// TIA Portal project "main" (V14)

(* hardware
DEVICE "GSD-Geraet_1"  GSD.Device.PN
   slot 0: "Baugruppenträger"  Rail  V1.0
   slot 0: "Station1"  BNI005H  V3.0
   slot 4: "SmartLight2"  IOL_I/O_08/08 byte
      slot 0: "IOL_I/O_08/08 byte"  IOL_I/O_08/08 byte
DEVICE "ET 200SP-Station_2"  ET 200SP-Station
   slot 0: "Baugruppenträger_0"  6ES5 710-8MAx1
   slot 1: "PLC_1"  CPU 1512SP F-1 PN  6ES7 512-1SK01-0AB0  V2.0
   slot 2: "DI 8x24VDC HF_1"  DI 8x24VDC HF  6ES7 131-6BF00-0CA0  V1.2
      slot 1: "DI 8x24VDC HF_1"  DI 8x24VDC HF
   slot 3: "Servermodul_1"  Servermodul  6ES7 193-6PA00-0AA0  V1.0
      slot 1: "Servermodul_1"  Servermodul
   slot 127: "BA 2xRJ45"  BA 2xRJ45  6ES7 193-6AR00-0AA0  V0.0
      slot 32769: "Port_1"  6ES7 193-6AR00-0AA0
      slot 32770: "Port_2"  6ES7 193-6AR00-0AA0
DEVICE "GSD-Geraet_2"  GSD.Device.PN
   slot 0: "Baugruppenträger"  Rail  V1.0
   slot 0: "Station2"  BNI005H  V3.0
DEVICE "GSD-Geraet_3"  GSD.Device.PN
   slot 0: "Baugruppenträger"  Rail  V1.0
   slot 0: "Station3"  BNI005H  V3.0
DEVICE "GSD-Geraet_4"  GSD.Device.PN
   slot 0: "Baugruppenträger"  Rail  V1.0
   slot 0: "Station4"  BNI005H  V3.0
   slot 4: "IOL_I/O_16/16 byte_3"  IOL_I/O_16/16 byte
      slot 0: "IOL_I/O_16/16 byte"  IOL_I/O_16/16 byte
DEVICE "GSD-Geraet_5"  GSD.Device.PN
   slot 0: "Baugruppenträger"  Rail  V1.0
   slot 0: "Station6"  BNI005H  V3.0
DEVICE "GSD-Geraet_6"  GSD.Device.PN
   slot 0: "Baugruppenträger"  Rail  V1.0
   slot 0: "Station8"  BNI005H  V3.0
   slot 3: "IOL_I/O_16/16 byte_2"  IOL_I/O_16/16 byte
      slot 0: "IOL_I/O_16/16 byte"  IOL_I/O_16/16 byte
   slot 4: "SmartLight"  IOL_I/O_08/08 byte
      slot 0: "IOL_I/O_08/08 byte"  IOL_I/O_08/08 byte
DEVICE "GSD-Geraet_7"  GSD.Device.PN
   slot 0: "Baugruppenträger"  Rail  V1.0
   slot 0: "Station7"  BNI005H  V3.0
DEVICE "GSD-Geraet_8"  GSD.Device.PN
   slot 0: "Baugruppenträger"  Rail  V1.0
   slot 0: "Station5"  BNI005H  V3.0
DEVICE "GSD-Geraet_9"  GSD.Device.PN
   slot 0: "Baugruppenträger"  Rail  V1.0
   slot 0: "Station10"  BNI005H  V3.0
DEVICE "GSD-Geraet_10"  GSD.Device.PN
   slot 0: "Baugruppenträger"  Rail  V1.0
   slot 0: "Station9"  BNI005H  V3.0
   slot 3: "IOL_I/O_16/16 byte_2"  IOL_I/O_16/16 byte
      slot 0: "IOL_I/O_16/16 byte"  IOL_I/O_16/16 byte
DEVICE "GSD-Geraet_11"  GSD.Device.PN
   slot 0: "Baugruppenträger"  Rail  V1.0
   slot 0: "Station11"  BNI005H  V3.0
   slot 4: "SmartLight2"  IOL_I/O_08/08 byte
      slot 0: "IOL_I/O_08/08 byte"  IOL_I/O_08/08 byte
DEVICE "GSD-Geraet_12"  GSD.Device.PN
   slot 0: "Baugruppenträger"  Rail  V1.0
   slot 0: "Station12"  BNI005H  V3.0
DEVICE "GSD-Geraet_13"  GSD.Device.PN
   slot 0: "Baugruppenträger"  Rail  V1.0
   slot 0: "Station13"  BNI005H  V3.0
DEVICE "GSD-Geraet_14"  GSD.Device.PN
   slot 0: "Baugruppenträger"  Rail  V1.0
   slot 0: "Station15"  BNI005H  V3.0
DEVICE "GSD-Geraet_15"  GSD.Device.PN
   slot 0: "Baugruppenträger"  Rail  V1.0
   slot 0: "Station16"  BNI005H  V3.0
DEVICE "GSD-Geraet_16"  GSD.Device.PN
   slot 0: "Baugruppenträger"  Rail  V1.0
   slot 0: "Station17"  BNI005H  V3.0
DEVICE "GSD-Geraet_17"  GSD.Device.PN
   slot 0: "Baugruppenträger"  Rail  V1.0
   slot 0: "Station20"  BNI005H  V3.0
DEVICE "GSD-Geraet_18"  GSD.Device.PN
   slot 0: "Baugruppenträger"  Rail  V1.0
   slot 0: "Station19"  BNI005H  V3.0
   slot 3: "IOL_I/O_16/16 byte_2"  IOL_I/O_16/16 byte
      slot 0: "IOL_I/O_16/16 byte"  IOL_I/O_16/16 byte
DEVICE "GSD-Geraet_19"  GSD.Device.PN
   slot 0: "Baugruppenträger"  Rack  V1.0
   slot 0: "BVS-SC"  BVS-SC  BVS_SC  V1.x
      slot 0: "BVS-SC"  BVS-SC
      slot 1: "PN-IO"  PN-IO
         slot 1: "port 1 - M12"  port 1 - M12
   slot 1: "SmartCamera E/A 128/16 Byte_1"  SmartCamera I/O 128/16 byte
      slot 0: "SmartCamera E/A 128/16 Byte"  SmartCamera I/O 128/16 byte
*)

// ===== PLC "PLC_1"  CPU 1512SP F-1 PN =====

VAR_GLOBAL   // PLC tag table "Standard-Variablentabelle"
   "EingangM1P1" AT %I1001.0 : Bool;
   "ByteM1P1.1" AT %IB1002 : Byte;
   "ByteM1P1.2" AT %IB1003 : Byte;
   "ByteM1P1.3" AT %IB1004 : Byte;
   "ByteM1P1.4" AT %IB1005 : Byte;
   "ByteM1P1.5" AT %IB1006 : Byte;
   "ByteM1P1.6" AT %IB1007 : Byte;
   "ByteM1P1.7" AT %IB1008 : Byte;
   "ByteM1P1.8" AT %IB1009 : Byte;
   "ByteM2P1.1" AT %IB2002 : Byte;
   "ByteM2P1.2" AT %IB2003 : Byte;
   "ByteM2P1.3" AT %IB2004 : Byte;
   "ByteM2P1.4" AT %IB2005 : Byte;
   "ByteM2P1.5" AT %IB2006 : Byte;
   "ByteM2P1.6" AT %IB2007 : Byte;
   "ByteM2P1.7" AT %IB2008 : Byte;
   "ByteM2P1.8" AT %IB2009 : Byte;
   "EingangM2P1" AT %I2001.0 : Bool;
   "ByteM3P1.1" AT %IB3002 : Byte;
   "ByteM3P1.2" AT %IB3003 : Byte;
   "ByteM3P1.3" AT %IB3004 : Byte;
   "ByteM3P1.4" AT %IB3005 : Byte;
   "ByteM3P1.5" AT %IB3006 : Byte;
   "ByteM3P1.6" AT %IB3007 : Byte;
   "ByteM3P1.7" AT %IB3008 : Byte;
   "ByteM3P1.8" AT %IB3009 : Byte;
   "EingangM3P1" AT %I3001.0 : Bool;
   "ByteM4P1.1" AT %IB4002 : Byte;
   "ByteM4P1.2" AT %IB4003 : Byte;
   "ByteM4P1.3" AT %IB4004 : Byte;
   "ByteM4P1.4" AT %IB4005 : Byte;
   "ByteM4P1.5" AT %IB4006 : Byte;
   "ByteM4P1.6" AT %IB4007 : Byte;
   "ByteM4P1.7" AT %IB4008 : Byte;
   "ByteM4P1.8" AT %IB4009 : Byte;
   "EingangM4P1" AT %I4001.0 : Bool;
   "ByteM5P1.1" AT %IB5002 : Byte;
   "ByteM5P1.2" AT %IB5003 : Byte;
   "ByteM5P1.3" AT %IB5004 : Byte;
   "ByteM5P1.4" AT %IB5005 : Byte;
   "ByteM5P1.5" AT %IB5006 : Byte;
   "ByteM5P1.6" AT %IB5007 : Byte;
   "ByteM5P1.7" AT %IB5008 : Byte;
   "ByteM5P1.8" AT %IB5009 : Byte;
   "EingangM5P1" AT %I5001.0 : Bool;
   "ByteM6P1.1" AT %IB6002 : Byte;
   "ByteM6P1.2" AT %IB6003 : Byte;
   "ByteM6P1.3" AT %IB6004 : Byte;
   "ByteM6P1.4" AT %IB6005 : Byte;
   "ByteM6P1.5" AT %IB6006 : Byte;
   "ByteM6P1.6" AT %IB6007 : Byte;
   "ByteM6P1.7" AT %IB6008 : Byte;
   "ByteM6P1.8" AT %IB6009 : Byte;
   "EingangM6P1" AT %I6001.0 : Bool;
   "ByteM7P1.1" AT %IB7002 : Byte;
   "ByteM7P1.2" AT %IB7003 : Byte;
   "ByteM7P1.3" AT %IB7004 : Byte;
   "ByteM7P1.4" AT %IB7005 : Byte;
   "ByteM7P1.5" AT %IB7006 : Byte;
   "ByteM7P1.6" AT %IB7007 : Byte;
   "ByteM7P1.7" AT %IB7008 : Byte;
   "ByteM7P1.8" AT %IB7009 : Byte;
   "EingangM7P1" AT %I7001.0 : Bool;
   "ByteM8P1.1" AT %IB8002 : Byte;
   "ByteM8P1.2" AT %IB8003 : Byte;
   "ByteM8P1.3" AT %IB8004 : Byte;
   "ByteM8P1.4" AT %IB8005 : Byte;
   "ByteM8P1.5" AT %IB8006 : Byte;
   "ByteM8P1.6" AT %IB8007 : Byte;
   "ByteM8P1.7" AT %IB8008 : Byte;
   "ByteM8P1.8" AT %IB8009 : Byte;
   "EingangM8P1" AT %I8001.0 : Bool;
   "ByteM9P1.1" AT %IB9002 : Byte;
   "ByteM9P1.2" AT %IB9003 : Byte;
   "ByteM9P1.3" AT %IB9004 : Byte;
   "ByteM9P1.4" AT %IB9005 : Byte;
   "ByteM9P1.5" AT %IB9006 : Byte;
   "ByteM9P1.6" AT %IB9007 : Byte;
   "ByteM9P1.7" AT %IB9008 : Byte;
   "ByteM9P1.8" AT %IB9009 : Byte;
   "EingangM9P1" AT %I9001.0 : Bool;
   "ByteM10P1.1" AT %IB10002 : Byte;
   "ByteM10P1.2" AT %IB10003 : Byte;
   "ByteM10P1.3" AT %IB10004 : Byte;
   "ByteM10P1.4" AT %IB10005 : Byte;
   "ByteM10P1.5" AT %IB10006 : Byte;
   "ByteM10P1.6" AT %IB10007 : Byte;
   "ByteM10P1.7" AT %IB10008 : Byte;
   "ByteM10P1.8" AT %IB10009 : Byte;
   "EingangM10P1" AT %I10001.0 : Bool;
   "ByteM11P1.1" AT %IB11002 : Byte;
   "ByteM11P1.2" AT %IB11003 : Byte;
   "ByteM11P1.3" AT %IB11004 : Byte;
   "ByteM11P1.4" AT %IB11005 : Byte;
   "ByteM11P1.5" AT %IB11006 : Byte;
   "ByteM11P1.6" AT %IB11007 : Byte;
   "ByteM11P1.7" AT %IB11008 : Byte;
   "ByteM11P1.8" AT %IB11009 : Byte;
   "EingangM11P1" AT %I11001.0 : Bool;
   "ByteM12P1.1" AT %IB12002 : Byte;
   "ByteM12P1.2" AT %IB12003 : Byte;
   "ByteM12P1.3" AT %IB12004 : Byte;
   "ByteM12P1.4" AT %IB12005 : Byte;
   "ByteM12P1.5" AT %IB12006 : Byte;
   "ByteM12P1.6" AT %IB12007 : Byte;
   "ByteM12P1.7" AT %IB12008 : Byte;
   "ByteM12P1.8" AT %IB12009 : Byte;
   "EingangM12P1" AT %I12001.0 : Bool;
   "ByteM13P1.1" AT %IB13002 : Byte;
   "ByteM13P1.2" AT %IB13003 : Byte;
   "ByteM13P1.3" AT %IB13004 : Byte;
   "ByteM13P1.4" AT %IB13005 : Byte;
   "ByteM13P1.5" AT %IB13006 : Byte;
   "ByteM13P1.6" AT %IB13007 : Byte;
   "ByteM13P1.7" AT %IB13008 : Byte;
   "ByteM13P1.8" AT %IB13009 : Byte;
   "EingangM13P1" AT %I13001.0 : Bool;
   "ByteM15P1.1" AT %IB15002 : Byte;
   "ByteM15P1.2" AT %IB15003 : Byte;
   "ByteM15P1.3" AT %IB15004 : Byte;
   "ByteM15P1.4" AT %IB15005 : Byte;
   "ByteM15P1.5" AT %IB15006 : Byte;
   "ByteM15P1.6" AT %IB15007 : Byte;
   "ByteM15P1.7" AT %IB15008 : Byte;
   "ByteM15P1.8" AT %IB15009 : Byte;
   "EingangM15P1" AT %I15001.0 : Bool;
   "ByteM16P1.1" AT %IB16002 : Byte;
   "ByteM16P1.2" AT %IB16003 : Byte;
   "ByteM16P1.3" AT %IB16004 : Byte;
   "ByteM16P1.4" AT %IB16005 : Byte;
   "ByteM16P1.5" AT %IB16006 : Byte;
   "ByteM16P1.6" AT %IB16007 : Byte;
   "ByteM16P1.7" AT %IB16008 : Byte;
   "ByteM16P1.8" AT %IB16009 : Byte;
   "EingangM16P1" AT %I16001.0 : Bool;
   "ByteM17P1.1" AT %IB17002 : Byte;
   "ByteM17P1.2" AT %IB17003 : Byte;
   "ByteM17P1.3" AT %IB17004 : Byte;
   "ByteM17P1.4" AT %IB17005 : Byte;
   "ByteM17P1.5" AT %IB17006 : Byte;
   "ByteM17P1.6" AT %IB17007 : Byte;
   "ByteM17P1.7" AT %IB17008 : Byte;
   "ByteM17P1.8" AT %IB17009 : Byte;
   "EingangM17P1" AT %I17001.0 : Bool;
   "ByteM19P1.1" AT %IB19002 : Byte;
   "ByteM19P1.2" AT %IB19003 : Byte;
   "ByteM19P1.3" AT %IB19004 : Byte;
   "ByteM19P1.4" AT %IB19005 : Byte;
   "ByteM19P1.5" AT %IB19006 : Byte;
   "ByteM19P1.6" AT %IB19007 : Byte;
   "ByteM19P1.7" AT %IB19008 : Byte;
   "ByteM19P1.8" AT %IB19009 : Byte;
   "EingangM19P1" AT %I19001.0 : Bool;
   "ByteM20P1.1" AT %IB20002 : Byte;
   "ByteM20P1.2" AT %IB20003 : Byte;
   "ByteM20P1.3" AT %IB20004 : Byte;
   "ByteM20P1.4" AT %IB20005 : Byte;
   "ByteM20P1.5" AT %IB20006 : Byte;
   "ByteM20P1.6" AT %IB20007 : Byte;
   "ByteM20P1.7" AT %IB20008 : Byte;
   "ByteM20P1.8" AT %IB20009 : Byte;
   "EingangM20P1" AT %I20001.0 : Bool;
   "EingangM4P2" AT %I4017.0 : Bool;
   "EingangM8P2" AT %I8017.0 : Bool;
   "ByteM8P2.1" AT %IB8018 : Byte;
   "ByteM8P2.2" AT %IB8019 : Byte;
   "ByteM8P2.3" AT %IB8020 : Byte;
   "ByteM8P2.4" AT %IB8021 : Byte;
   "ByteM8P2.5" AT %IB8022 : Byte;
   "ByteM8P2.6" AT %IB8023 : Byte;
   "ByteM8P2.7" AT %IB8024 : Byte;
   "ByteM8P2.8" AT %IB8025 : Byte;
   "EingangM9P2" AT %I9017.0 : Bool;
   "ByteM9P2.1" AT %IB9018 : Byte;
   "ByteM9P2.2" AT %IB9019 : Byte;
   "ByteM9P2.3" AT %IB9020 : Byte;
   "ByteM9P2.4" AT %IB9021 : Byte;
   "ByteM9P2.5" AT %IB9022 : Byte;
   "ByteM9P2.6" AT %IB9023 : Byte;
   "ByteM9P2.7" AT %IB9024 : Byte;
   "ByteM9P2.8" AT %IB9025 : Byte;
   "EingangM19P2" AT %I19017.0 : Bool;
   "ByteM19P2.1" AT %IB19018 : Byte;
   "ByteM19P2.2" AT %IB19019 : Byte;
   "ByteM19P2.3" AT %IB19020 : Byte;
   "ByteM19P2.4" AT %IB19021 : Byte;
   "ByteM19P2.5" AT %IB19022 : Byte;
   "ByteM19P2.6" AT %IB19023 : Byte;
   "ByteM19P2.7" AT %IB19024 : Byte;
   "ByteM19P2.8" AT %IB19025 : Byte;
   "EingangM4P2_AE" AT %I4017.2 : Bool;
   "EingangM4P3" AT %I4033.0 : Bool;
   "OutByteM1P2.1" AT %QB1017 : Byte;
   "BuzzerSmLi1" AT %Q1019.7 : Bool;
   "OutByteM4P2.1" AT %QB4018 : Byte;
   "OutHeader1M4P2_AV" AT %Q4017.0 : Bool;
   "OutByteM4P2.8" AT %QB4025 : Byte;
   "OutByteM4P2.7" AT %QB4024 : Byte;
   "OutByteM4P2.6" AT %QB4023 : Byte;
   "OutByteM4P2.5" AT %QB1022 : Byte;
   "OutByteM4P2.4" AT %QB4021 : Byte;
   "OutByteM4P2.3" AT %QB4020 : Byte;
   "OutByteM4P2.2" AT %QB4019 : Byte;
   "OutHeader2M4P2_AV" AT %Q4026.0 : Bool;
   "OutByteM1P3_Level8bit" AT %QB1027 : Byte;
   "SmLiS1P3-0.0" AT %Q1021.0 : Bool;
   "SmLiS1P3-0.1" AT %Q1021.1 : Bool;
   "SmLiS1P3-0.2" AT %Q1021.2 : Bool;
   "SmLiS1P3-0.3" AT %Q1021.3 : Bool;
   "SmLiS1P3-0.4" AT %Q1021.4 : Bool;
   "SmLiS1P3-0.5" AT %Q1021.5 : Bool;
   "SmLiS1P3-0.6" AT %Q1021.6 : Bool;
   "SmLiS1P3-0.7" AT %Q1021.7 : Bool;
   "SmLiS1P3-1.0" AT %Q1022.0 : Bool;
   "SmLiS1P3-1.1" AT %Q1022.1 : Bool;
   "SmLiS1P3-1.3" AT %Q1022.3 : Bool;
   "SmLiS1P3-1.4" AT %Q1022.4 : Bool;
   "SmLiS1P3-1.5" AT %Q1022.5 : Bool;
   "SmLiS1P3-1.6" AT %Q1022.6 : Bool;
   "SmLiS1P3-1.2" AT %Q1022.2 : Bool;
   "SmLiS1P3-1.7" AT %Q1022.7 : Bool;
   "SmLiS1P3-2.3" AT %Q1023.3 : Bool;
   "SmLiS1P3-2.2" AT %Q1023.2 : Bool;
   "SmLiS1P3-2.1" AT %Q1023.1 : Bool;
   "SmLiS1P3-2.0" AT %Q1023.0 : Bool;
   "SmLiS1P3-3.1-Levelmode" AT %Q1024.1 : Bool;
   "OutByteM11P2.1" AT %QB11017 : Byte;
   "OutByteM11P3_Level8bit" AT %QB11027 : Byte;
   "SmLiS11P3-0.0" AT %Q11021.0 : Bool;
   "SmLiS11P3-0.1" AT %Q11021.1 : Bool;
   "SmLiS11P3-0.2" AT %Q11021.2 : Bool;
   "SmLiS11P3-0.3" AT %Q11021.3 : Bool;
   "SmLiS11P3-0.4" AT %Q11021.4 : Bool;
   "SmLiS11P3-0.5" AT %Q11021.5 : Bool;
   "SmLiS11P3-0.6" AT %Q11021.6 : Bool;
   "SmLiS11P3-0.7" AT %Q11021.7 : Bool;
   "SmLiS11P3-1.0" AT %Q11022.0 : Bool;
   "SmLiS11P3-1.1" AT %Q11022.1 : Bool;
   "SmLiS11P3-1.2" AT %Q11022.2 : Bool;
   "SmLiS11P3-1.3" AT %Q11022.3 : Bool;
   "SmLiS11P3-1.4" AT %Q11022.4 : Bool;
   "SmLiS11P3-1.5" AT %Q11022.5 : Bool;
   "SmLiS11P3-1.6" AT %Q11022.6 : Bool;
   "SmLiS11P3-1.7" AT %Q11022.7 : Bool;
   "SmLiS11P3-2.0" AT %Q11023.0 : Bool;
   "SmLiS11P3-2.1" AT %Q11023.1 : Bool;
   "SmLiS11P3-2.2" AT %Q11023.2 : Bool;
   "SmLiS11P3-2.3" AT %Q11023.3 : Bool;
   "SmLiS11P3-3.1-Levelmode" AT %Q11024.1 : Bool;
   "SmLiS8P3-0.0" AT %Q8033.0 : Bool;
   "SmLiS8P3-0.1" AT %Q8033.1 : Bool;
   "SmLiS8P3-0.4" AT %Q8033.4 : Bool;
   "SmLiS8P3-0.5" AT %Q8033.5 : Bool;
   "SmLiS8P3-1.0" AT %Q8034.0 : Bool;
   "SmLiS8P3-1.1" AT %Q8034.1 : Bool;
   "SmLiS8P3-1.4" AT %Q8034.4 : Bool;
   "SmLiS8P3-1.5" AT %Q8034.5 : Bool;
   "SmLiS8P3-2.0" AT %Q8035.0 : Bool;
   "SmLiS8P3-2.1" AT %Q8035.1 : Bool;
   "SmLiS8P3-3.0-Segmentmode" AT %Q8036.0 : Bool;
   "Clock" AT %M0.0 : Bool;
   "inPuffer" AT %MB100 : Byte;
   "ausPuffer" AT %MB2 : Byte;
   "Testmerker1" AT %M0.1 : Bool;
   "SC_CommandStart" AT %M0.2 : Bool;
   "SC_CamResetWarn" AT %M200.0 : Bool;
   "SC_GetResults" AT %M0.7 : Bool;
   "SC_Trigger" AT %M0.6 : Bool;
   "SC_StartRun" AT %M0.5 : Bool;
   "SC_StopRun" AT %M0.4 : Bool;
   "SC_ResetWarnings" AT %M0.3 : Bool;
   "MerkerCommandSC" AT %MW201 : Int;
   "S9P1IB0.2_AE" AT %I9001.2 : Bool;
   "S9P1IB0.1_AA" AT %I9001.1 : Bool;
   "S9P1OB0.0_AV" AT %Q9001.0 : Bool;
   "S9P1OB1_CommandDesignator" AT %QB9002 : Byte;
   "S9P1OB2_StartAdressLow" AT %QB9003 : Byte;
   "S9P1OB3_StartAdressHigh" AT %QB9004 : Byte;
   "S9P1OB4_NumBytesLow" AT %QB9005 : Byte;
   "S9P1OB5_NumBytesHigh" AT %QB9006 : Byte;
   "S9P1OB9.0_AV" AT %Q9010.0 : Bool;
   "S1P1OB1_CommandDesignator" AT %QB1002 : Byte;
   "S1P1OB2_StartAdressLow" AT %QB1003 : Byte;
   "S1P1OB3_StartAdressHigh" AT %QB1004 : Byte;
   "S1P1OB4_NumBytesLow" AT %QB1005 : Byte;
   "S1P1OB4_NumBytesHigh" AT %QB1006 : Byte;
   "S1P1OB0.0_AV" AT %Q1001.0 : Bool;
   "S1P1OB9.0_AV" AT %Q1010.0 : Bool;
   "S1P1IB0.2_AE" AT %Q1010.2 : Bool;
   "S1P1IB0.3_AF" AT %Q1010.3 : Bool;
   "S1P1IB0.1_AA" AT %Q1010.1 : Bool;
   "S9P2OB1_CommandDesignator" AT %QB9018 : Byte;
   "S9P2OB2_StartAdressLow" AT %QB9019 : Byte;
   "S9P2OB3_StartAdressHigh" AT %QB9020 : Byte;
   "S9P2OB4_NumBytesLow" AT %QB9021 : Byte;
   "S9P2OB4_NumBytesHigh" AT %QB9022 : Byte;
   "S9P2OB0.0_AV" AT %Q9017.0 : Bool;
   "S9P2OB9.0_AV" AT %Q9026.0 : Bool;
   "S9P2IB0.2_AE" AT %Q9017.2 : Bool;
   "S9P2IB0.3_AF" AT %Q9017.3 : Bool;
   "S9P2IB0.1_AA" AT %Q9017.1 : Bool;
   "ByteM4P2.1" AT %IB4018 : Byte;
   "ByteM4P2.2" AT %IB4019 : Byte;
   "ByteM4P2.3" AT %IB4020 : Byte;
   "ByteM4P2.4" AT %IB4021 : Byte;
   "ByteM4P2.5" AT %IB4022 : Byte;
   "ByteM4P2.6" AT %IB4023 : Byte;
   "ByteM4P2.7" AT %IB4024 : Byte;
   "ByteM4P2.8" AT %IB4025 : Byte;
   "ByteM4P3.1" AT %IB4034 : Byte;
   "ByteM4P3.2" AT %IB4035 : Byte;
   "ByteM4P3.3" AT %IB4036 : Byte;
   "ByteM4P3.4" AT %IB4037 : Byte;
   "ByteM4P3.5" AT %IB4038 : Byte;
   "ByteM4P3.6" AT %IB4039 : Byte;
   "ByteM4P3.7" AT %IB4040 : Byte;
   "ByteM4P3.8" AT %IB4041 : Byte;
   "Tag_1" AT %T1 : Timer;
END_VAR

DATA_BLOCK "IO_LINK_MASTER_DB"   // DB1
{ S7_Optimized_Access := 'TRUE' }
AUTHOR : Siemens
FAMILY : IO-Link
VERSION : 1.0
// stored: InstanceOfName IO_LINK_MASTER
"IO_LINK_MASTER"
BEGIN
END_DATA_BLOCK

DATA_BLOCK "IO_LINK_DEVICE_DB"   // DB2
{ S7_Optimized_Access := 'TRUE' }
AUTHOR : SUP_FA
FAMILY : IO-Link
VERSION : 3.0
// stored: InstanceOfName IO_LINK_DEVICE
"IO_LINK_DEVICE"
BEGIN
   write.data[0] := 16#03;
END_DATA_BLOCK

DATA_BLOCK "BVS_SC_DB"   // DB7
{ S7_Optimized_Access := 'TRUE' }
AUTHOR : BI-CU
FAMILY : Balluff
VERSION : 1.1
// stored: InstanceOfName BVS_SC
"BVS_SC"
BEGIN
END_DATA_BLOCK

DATA_BLOCK "00TEMP"   // DB8
{ S7_Optimized_Access := 'TRUE' }
VERSION : 0.1
   VAR
      EingriffPufferstand : Int;
      EingriffSmLiNummer : Int := 1;
      FlagEingriff : Bool;
      FlankenmerkerEingriff : Bool;
      Station1Umschaltung : Bool;
      TempAdresseFlag : Bool;
      RET_VAL : Int;
      PIADDR : UDInt;
      PICOUNT : UInt;
      PQADDR : UDInt;
      PQCOUNT : UInt;
      TempFlagPeek : Bool;
      ArrayTemp : Array[0..7] of Byte;
      ID : String;
      TempFlankenmerkePeek : Bool;
   END_VAR
BEGIN
END_DATA_BLOCK

DATA_BLOCK "FB35_Station1"   // DB11
{ S7_Optimized_Access := 'FALSE' }
AUTHOR : Serrano
FAMILY : Ident
NAME : BISM_IOL
VERSION : 1.0
// stored: InstanceOfName FB35_IOL_10Byte
"FB35_IOL_10Byte"
BEGIN
   Watchdog := S5T#3000MS;
END_DATA_BLOCK

DATA_BLOCK "Daten_zu_SC_Station8"   // DB12
{ S7_Optimized_Access := 'FALSE' }
VERSION : 0.1
   VAR
      SendByte : Array[0..99] of Byte;
   END_VAR
BEGIN
   SendByte[0] := 16#2;
   SendByte[1] := 16#0;
   SendByte[2] := 16#0;
   SendByte[3] := 16#0;
   SendByte[4] := 16#0;
END_DATA_BLOCK

DATA_BLOCK "Daten_von_SC_Station8"   // DB13
{ S7_Optimized_Access := 'FALSE' }
VERSION : 0.1
   VAR
      "n.u." : Byte;
      AppID : Byte;
      Buerstentraeger : Bool;
      "n.u._7" : Bool;
      "n.u._6" : Bool;
      "n.u._5" : Bool;
      "n.u._4" : Bool;
      "n.u._3" : Bool;
      "n.u._2" : Bool;
      "n.u._1" : Bool;
      GehaeuseUnten_Schraube : Bool;
      "n.u._14" : Bool;
      "n.u._13" : Bool;
      "n.u._12" : Bool;
      "n.u._11" : Bool;
      "n.u._10" : Bool;
      "n.u._9" : Bool;
      "n.u._8" : Bool;
      Zahnrad_klein : Bool;
      "n.u._21" : Bool;
      "n.u._20" : Bool;
      "n.u._19" : Bool;
      "n.u._18" : Bool;
      "n.u._17" : Bool;
      "n.u._16" : Bool;
      "n.u._15" : Bool;
      Zahnrad_gross : Bool;
      "n.u._28" : Bool;
      "n.u._27" : Bool;
      "n.u._26" : Bool;
      "n.u._25" : Bool;
      "n.u._24" : Bool;
      "n.u._23" : Bool;
      "n.u._22" : Bool;
      GehaeuseOben : Bool;
   END_VAR
BEGIN
END_DATA_BLOCK

DATA_BLOCK "DB_Ausfall_IO"   // DB16
{ S7_Optimized_Access := 'TRUE' }
VERSION : 0.1
   VAR
      ErrorCode_RD_SINFO : Int;
      ErrorCode_RD_SYS_T : Int;
      ErrorCode_LOG2GEO : Int;
      ErrorCode_D_ACT_DP : Int;
      ErrorCode_ModuleStates1 : Int;
      ErrorCode_ModuleStates2 : Int;
      StateBusy_D_ACT_DP : Bool;
      State1 : Array[0..127] of Bool;
      State2 : Array[0..127] of Bool;
      TimeOfEvent : DTL;
      FlagAdresseUmgewandelt : Bool;
      Info : SI_StationFailure;
      TempAdresse : Hw_Device;
      Info_2 : SI_classic;
      AdresseAusfall : GEOADDR;
      CounterS1 : Int;
      CounterS2 : Int;
      CounterS3 : Int;
      CounterS4 : Int;
      CounterS5 : Int;
      CounterS6 : Int;
      CounterS7 : Int;
      CounterS8 : Int;
      CounterS9 : Int;
      CounterS10 : Int;
      FlagDeaktivieren : Bool;
      bibop : Bool;
      ToggleNeu : Bool;
      CounterRack : Int;
      CounterStatus : Int;
      CounterProfile : Int;
      CounterPull : Int;
      CounterIO : Int;
      Adressen : Array[0..2] of HW_IO;
   END_VAR
BEGIN
END_DATA_BLOCK

DATA_BLOCK "Daten_von_SLK"   // DB17
{ S7_Optimized_Access := 'TRUE' }
VERSION : 0.1
   VAR
      V34 : Byte;
      V35 : Byte;
      V3 : Byte;
      V4 : Byte;
      V5 : Byte;
      V6 : Byte;
      V7 : Byte;
      V8 : Byte;
      V9 : Byte;
      V10 : Byte;
      V11 : Byte;
      V33 : Byte;
      V32 : Byte;
      V31 : Byte;
      V30 : Byte;
      V29 : Byte;
      V28 : Byte;
      V27 : Byte;
      V26 : Byte;
      V25 : Byte;
      V24 : Byte;
      V23 : Byte;
      V22 : Byte;
      V21 : Byte;
      V20 : Byte;
      V19 : Byte;
      V18 : Byte;
      V17 : Byte;
      V16 : Byte;
      V15 : Byte;
      V14 : Byte;
      V13 : Byte;
      V12 : Byte;
   END_VAR
BEGIN
END_DATA_BLOCK

DATA_BLOCK "Daten_zu_SLK"   // DB18
{ S7_Optimized_Access := 'TRUE' }
VERSION : 0.1
   VAR
      V11 : Byte;
      V34 : Byte;
      V33 : Byte;
      V32 : Byte;
      V31 : Byte;
      V30 : Byte;
      V29 : Byte;
      V28 : Byte;
      V27 : Byte;
      V26 : Byte;
      V25 : Byte;
      V24 : Byte;
      V23 : Byte;
      V22 : Byte;
      V21 : Byte;
      V20 : Byte;
      V19 : Byte;
      V18 : Byte;
      V17 : Byte;
      V16 : Byte;
      V15 : Byte;
      V14 : Byte;
      V13 : Byte;
      V12 : Byte;
   END_VAR
BEGIN
END_DATA_BLOCK

DATA_BLOCK "Lese_DB_1"   // DB19
{ S7_Optimized_Access := 'TRUE' }
VERSION : 0.1
// stored: InstanceOfName Lese
"Lese"
BEGIN
   Adresse := 1002;
   EndeAdresse := 1009;
END_DATA_BLOCK

DATA_BLOCK "DB_Konstanten"   // DB20
{ S7_Optimized_Access := 'TRUE' }
VERSION : 0.1
   VAR
      HW_Adressen : Array[0..19] of HW_ANY;
      "Anzahl Adressen" : Int := 20;
      DEFAULT_STATION4_MAXPUFFER : Array[0..1] of Int;
   END_VAR
BEGIN
   DEFAULT_STATION4_MAXPUFFER[1] := 19;
   DEFAULT_STATION4_MAXPUFFER[0] := 12;
END_DATA_BLOCK

DATA_BLOCK "Test"   // DB21
{ S7_Optimized_Access := 'TRUE' }
VERSION : 0.1
   VAR
      RetValD_ACT_DP2 : Int;
      RetValD_ACT_DP1 : Int;
      RetValD_ACT_DP3 : Int;
      RetValState1 : Int;
      RetValState2 : Int;
      Busy1 : Bool;
      Busy2 : Bool;
      Busy3 : Bool;
      State1 : Bool;
      State2 : Bool;
      Req : Bool;
      IstDeakt1 : Int;
      IstDeakt2 : Int;
      FlagDeak : Bool;
      FlagDeakAll1 : Bool;
      FlagDeakAll2 : Bool;
      FlagDeakAll3 : Bool;
      FlagDeakAll4 : Bool;
      FlagDeakAll5 : Bool;
      FlagAk : Bool;
   END_VAR
BEGIN
END_DATA_BLOCK

DATA_BLOCK "DB_Station1_Port1"   // DB101
{ S7_Optimized_Access := 'FALSE' }
VERSION : 0.1
   VAR
      TagAtHead : Bool;
      Station : Byte := 1;
      Port : Byte := 1;
      CurrentValue_ULInt : ULInt;
      CurrentValue : String;
      RET_VAL : Int := 0;
      Busy : Bool := false;
      Deactivated : Bool := false;
      State : Bool;
      State2 : Bool;
      RET_VAL_module_state : Int;
      IDRead : Bool;
      PoltopfLength : Byte;
      Flag : Bool;
      Done : Bool;
      TimeWaited : Time;
      TempFlagDeaktivierung : Bool;
      TEMPCounter : Int;
      S1P1FlankePos : Bool;
   END_VAR
BEGIN
END_DATA_BLOCK

DATA_BLOCK "DB_Station2_Port1"   // DB201
{ S7_Optimized_Access := 'FALSE' }
VERSION : 0.1
   VAR
      TagAtHead : Bool;
      Station : Byte := 2;
      Port : Byte := 1;
      CurrentValue_ULInt : ULInt := 0;
      CurrentValue : String := '';
      RET_VAL : Int := 0;
      Busy : Bool := false;
      Deactivated : Bool := false;
      State : Bool;
      State2 : Bool;
      RET_VAL_module_state : Int;
   END_VAR
BEGIN
END_DATA_BLOCK

DATA_BLOCK "DB_Station3_Port1"   // DB301
{ S7_Optimized_Access := 'FALSE' }
VERSION : 0.1
   VAR
      TagAtHead : Bool;
      Station : Byte := 3;
      Port : Byte := 1;
      CurrentValue_ULInt : ULInt := 0;
      CurrentValue : String := '';
      RET_VAL : Int := 0;
      Busy : Bool := false;
      Deactivated : Bool := false;
      State : Bool;
      State2 : Bool;
      RET_VAL_module_state : Int;
   END_VAR
BEGIN
END_DATA_BLOCK

DATA_BLOCK "DB_Station4_Port1"   // DB401
{ S7_Optimized_Access := 'FALSE' }
VERSION : 0.1
   VAR
      TagAtHead : Bool;
      Station : Byte := 4;
      Port : Byte := 1;
      CurrentValue_ULInt : ULInt := 0;
      CurrentValue : String := '';
      LastValue_ULInt : ULInt := 0;
      RET_VAL : Int := 0;
      Busy : Bool := false;
      Deactivated : Bool := false;
      State : Bool;
      State2 : Bool;
      RET_VAL_module_state : Int;
   END_VAR
BEGIN
END_DATA_BLOCK

DATA_BLOCK "DB_Station4_Puffer"   // DB410
{ S7_Optimized_Access := 'FALSE' }
VERSION : 0.1
   VAR
      CONST_MAXPUFFER : Array[0..1] of Int;
      CONST_STARTWERT_SMLI1 : Int := 0;
      Pufferstand : Array[0..1] of Int;
      Faktoren : Array[0..1] of Int;
      CurrentID1 : ULInt;
      LastID1 : ULInt;
      CurrentID2 : ULInt;
      LastID2 : ULInt;
      TimeRun1 : Time := T#5s;
      TimeRun2 : Time;
      FlankenmerkerPort1Pos : Bool;
      FlankenmerkerPort2Neg : Bool;
      FlankenmerkerPort3Neg : Bool;
      FlankenmerkerPort2Pos : Bool;
      FlankenmerkerPort3Pos : Bool;
      FlankenmerkerPosTime1 : Bool;
      FlankenmerkerPosTime2 : Bool;
      FlagTimerStart1 : Bool;
      FlagTimerStart2 : Bool;
      FlagShortcut1 : Bool;
      FlagShortcut2 : Bool;
      temp : Bool;
   END_VAR
BEGIN
   CONST_MAXPUFFER[0] := 12;
   CONST_MAXPUFFER[1] := 19;
   Faktoren[0] := 0;
   Faktoren[1] := 0;
END_DATA_BLOCK

DATA_BLOCK "DB_Station5_Port1"   // DB501
{ S7_Optimized_Access := 'FALSE' }
VERSION : 0.1
   VAR
      TagAtHead : Bool;
      Station : Byte := 5;
      Port : Byte := 1;
      CurrentValue_ULInt : ULInt := 0;
      CurrentValue : String := '';
      RET_VAL : Int := 0;
      Busy : Bool := false;
      Deactivated : Bool := false;
      State : Bool;
      State2 : Bool;
      RET_VAL_module_state : Int;
   END_VAR
BEGIN
END_DATA_BLOCK

DATA_BLOCK "DB_Station6_Port1"   // DB601
{ S7_Optimized_Access := 'FALSE' }
VERSION : 0.1
   VAR
      TagAtHead : Bool;
      Station : Byte := 6;
      Port : Byte := 1;
      CurrentValue_ULInt : ULInt := 0;
      CurrentValue : String := '';
      RET_VAL : Int := 0;
      Busy : Bool := false;
      Deactivated : Bool := false;
      State : Bool;
      State2 : Bool;
      RET_VAL_module_state : Int;
   END_VAR
BEGIN
END_DATA_BLOCK

DATA_BLOCK "DB_Station7_Port1"   // DB701
{ S7_Optimized_Access := 'FALSE' }
VERSION : 0.1
   VAR
      TagAtHead : Bool;
      Station : Byte := 7;
      Port : Byte := 1;
      CurrentValue_ULInt : ULInt := 0;
      CurrentValue : String := '';
      RET_VAL : Int := 0;
      Busy : Bool := false;
      Deactivated : Bool := false;
      State : Bool;
      State2 : Bool;
      RET_VAL_module_state : Int;
   END_VAR
BEGIN
END_DATA_BLOCK

DATA_BLOCK "DB_Station8_Port1"   // DB801
{ S7_Optimized_Access := 'FALSE' }
VERSION : 0.1
   VAR
      TagAtHead : Bool;
      Station : Byte := 8;
      Port : Byte := 1;
      CurrentValue_ULInt : ULInt := 0;
      CurrentValue : String := '';
      RET_VAL : Int := 0;
      RET_VAL_Camera : Int;
      Busy_Camera : Bool;
      Busy : Bool := false;
      Deactivated : Bool := false;
      State : Bool;
      State2 : Bool;
      RET_VAL_module_state : Int;
   END_VAR
BEGIN
END_DATA_BLOCK

DATA_BLOCK "DB_Station8_Port2"   // DB802
{ S7_Optimized_Access := 'FALSE' }
VERSION : 0.1
   VAR
      TagAtHead : Bool;
      Station : Byte := 8;
      Port : Byte := 2;
      CurrentValue_ULInt : ULInt := 0;
      CurrentValue : String := '';
   END_VAR
BEGIN
END_DATA_BLOCK

DATA_BLOCK "DB_SC_Station8"   // DB810
{ S7_Optimized_Access := 'TRUE' }
VERSION : 0.1
   VAR
      Buerstentraeger : Bool;
      GehaeuseUnten_Schraube : Bool;
      Zahnrad_klein : Bool;
      Zahnrad_gross : Bool;
      GehaeuseOben : Bool;
      FlankenmerkerP1 : Bool;
      FlankenmerkerP4 : Bool;
      FlankenmerkerP3 : Bool;
      FlankenmerkerP2 : Bool;
      FlankenmerkerGetResult1 : Bool;
      FlankenmerkerGetResult2 : Bool;
      setzezurüeck1 : Bool;
      setzezurüeck2 : Bool;
      startePruefung : Bool;
      CommandFlanke1 : Bool;
      StartRun_Flanke : Bool;
      ResetWarnings_Flanke : Bool;
      StopRun_Flanke : Bool;
      GetResult_Flanke : Bool;
      Trigger_Flanke : Bool;
      CamBusy_Flanke : Bool;
      Verzoegerung : Time;
   END_VAR
BEGIN
END_DATA_BLOCK

DATA_BLOCK "DB_Station9_Port1"   // DB901
{ S7_Optimized_Access := 'FALSE' }
VERSION : 0.1
   VAR
      TagAtHead : Bool;
      Station : Byte := 9;
      Port : Byte := 1;
      CurrentValue_ULInt : ULInt := 0;
      CurrentValue : String := '';
      RET_VAL : Int := 0;
      Busy : Bool := false;
      Deactivated : Bool := false;
      State : Bool;
      State2 : Bool;
      RET_VAL_module_state : Int;
      TriggerAltNeu : Bool := true;
      ToReadStartByteHigh : Byte := 16#0;
      ToReadStartByteLow : Byte;
      ToReadNumBytesLow : Byte := 16#1;
      ToReadNumBytesHigh : Byte;
      ReadByte1 : Byte := 16#27;
      ReadByte2 : Byte := 16#27;
      ReadByte3 : Byte := 16#27;
      ReadByte4 : Byte := 16#27;
      ReadByte5 : Byte := 16#27;
      ReadByte6 : Byte := 16#27;
      ReadByte7 : Byte := 16#27;
      ReadByte8 : Byte := 16#27;
      ErrorCode : Byte;
      FlagAngekommen_4 : Bool;
      FlagAngekommen_3 : Bool;
      FlagAngekommen_2 : Bool;
      FlagAngekommen_1 : Bool;
      FlagAngekommen : Bool;
   END_VAR
BEGIN
END_DATA_BLOCK

DATA_BLOCK "DB_Station9_Port2"   // DB902
{ S7_Optimized_Access := 'FALSE' }
VERSION : 0.1
   VAR
      TagAtHead : Bool;
      Station : Byte := 9;
      Port : Byte := 2;
      CurrentValue_ULInt : ULInt := 0;
      CurrentValue : String := '';
      IDRead : Bool;
      PoltopfLength : Byte;
      Flag : Bool;
      Done : Bool;
      TimeWaited : Time;
   END_VAR
BEGIN
END_DATA_BLOCK

DATA_BLOCK "DB_Station10_Port1"   // DB1001
{ S7_Optimized_Access := 'FALSE' }
VERSION : 0.1
   VAR
      TagAtHead : Bool;
      Station : Byte := 10;
      Port : Byte := 1;
      CurrentValue_ULInt : ULInt := 0;
      CurrentValue : String := '';
      RET_VAL : Int := 0;
      Busy : Bool := false;
      Deactivated : Bool := false;
      State : Bool;
      State2 : Bool;
      RET_VAL_module_state : Int;
   END_VAR
BEGIN
END_DATA_BLOCK

DATA_BLOCK "DB_Station11_Port1"   // DB1101
{ S7_Optimized_Access := 'FALSE' }
VERSION : 0.1
   VAR
      TagAtHead : Bool;
      Station : Byte := 11;
      Port : Byte := 1;
      CurrentValue_ULInt : ULInt := 0;
      CurrentValue : String := '';
      RET_VAL : Int := 0;
      Busy : Bool := false;
      Deactivated : Bool := false;
      State : Bool;
      State2 : Bool;
      RET_VAL_module_state : Int;
   END_VAR
BEGIN
END_DATA_BLOCK

DATA_BLOCK "DB_Station12_Port1"   // DB1201
{ S7_Optimized_Access := 'FALSE' }
VERSION : 0.1
   VAR
      TagAtHead : Bool;
      Station : Byte := 12;
      Port : Byte := 1;
      CurrentValue_ULInt : ULInt := 0;
      CurrentValue : String := '';
      RET_VAL : Int := 0;
      Busy : Bool := false;
      Deactivated : Bool := false;
      State : Bool;
      State2 : Bool;
      RET_VAL_module_state : Int;
   END_VAR
BEGIN
END_DATA_BLOCK

DATA_BLOCK "DB_Station13_Port1"   // DB1301
{ S7_Optimized_Access := 'FALSE' }
VERSION : 0.1
   VAR
      TagAtHead : Bool;
      Station : Byte := 13;
      Port : Byte := 1;
      CurrentValue_ULInt : ULInt := 0;
      CurrentValue : String := '';
      RET_VAL : Int := 0;
      Busy : Bool := false;
      Deactivated : Bool := false;
      State : Bool;
      State2 : Bool;
      RET_VAL_module_state : Int;
   END_VAR
BEGIN
END_DATA_BLOCK

DATA_BLOCK "DB_Station15_Port1"   // DB1501
{ S7_Optimized_Access := 'FALSE' }
VERSION : 0.1
   VAR
      TagAtHead : Bool;
      Station : Byte := 15;
      Port : Byte := 1;
      CurrentValue_ULInt : ULInt := 0;
      CurrentValue : String := '';
      RET_VAL : Int := 0;
      Busy : Bool := false;
      Deactivated : Bool := false;
      State : Bool;
      State2 : Bool;
      RET_VAL_module_state : Int;
   END_VAR
BEGIN
END_DATA_BLOCK

DATA_BLOCK "DB_Station16_Port1"   // DB1601
{ S7_Optimized_Access := 'FALSE' }
VERSION : 0.1
   VAR
      TagAtHead : Bool;
      Station : Byte := 16;
      Port : Byte := 1;
      CurrentValue_ULInt : ULInt := 0;
      CurrentValue : String := '';
      RET_VAL : Int := 0;
      Busy : Bool := false;
      Deactivated : Bool := false;
      State : Bool;
      State2 : Bool;
      RET_VAL_module_state : Int;
   END_VAR
BEGIN
END_DATA_BLOCK

DATA_BLOCK "DB_Station17_Port1"   // DB1701
{ S7_Optimized_Access := 'FALSE' }
VERSION : 0.1
   VAR
      TagAtHead : Bool;
      Station : Byte := 17;
      Port : Byte := 1;
      CurrentValue_ULInt : ULInt := 0;
      CurrentValue : String := '';
      RET_VAL : Int := 0;
      Busy : Bool := false;
      Deactivated : Bool := false;
      State : Bool;
      State2 : Bool;
      RET_VAL_module_state : Int;
   END_VAR
BEGIN
END_DATA_BLOCK

DATA_BLOCK "DB_Station19_Port1"   // DB1901
{ S7_Optimized_Access := 'FALSE' }
VERSION : 0.1
   VAR
      TagAtHead : Bool;
      Station : Byte := 19;
      Port : Byte := 1;
      CurrentValue_ULInt : ULInt := 0;
      CurrentValue : String := '';
      RET_VAL : Int := 0;
      Busy : Bool := false;
      Deactivated : Bool := false;
      State : Bool;
      State2 : Bool;
      RET_VAL_module_state : Int;
   END_VAR
BEGIN
END_DATA_BLOCK

DATA_BLOCK "DB_Station19_Port2"   // DB1902
{ S7_Optimized_Access := 'FALSE' }
VERSION : 0.1
   VAR
      TagAtHead : Bool;
      Station : Byte := 19;
      Port : Byte := 2;
      CurrentValue_ULInt : ULInt := 0;
      CurrentValue : String := '';
   END_VAR
BEGIN
END_DATA_BLOCK

DATA_BLOCK "DB_Station20_Port1"   // DB2001
{ S7_Optimized_Access := 'FALSE' }
VERSION : 0.1
   VAR
      TagAtHead : Bool;
      Station : Byte := 20;
      Port : Byte := 1;
      CurrentValue_ULInt : ULInt := 0;
      CurrentValue : String := '';
      RET_VAL : Int := 0;
      Busy : Bool := false;
      Deactivated : Bool := false;
      State : Bool;
      State2 : Bool;
      RET_VAL_module_state : Int;
   END_VAR
BEGIN
END_DATA_BLOCK

// folder: System blocks/Program resources

DATA_BLOCK "TempTimer"   // DB3
{ S7_Optimized_Access := 'TRUE' }
AUTHOR : Simatic
FAMILY : IEC
NAME : IEC_TMR
VERSION : 1.0
// stored: InstanceOfName IEC_TIMER
"IEC_TIMER"
BEGIN
END_DATA_BLOCK

DATA_BLOCK "TempTimer2"   // DB4
{ S7_Optimized_Access := 'TRUE' }
AUTHOR : Simatic
FAMILY : IEC
NAME : IEC_TMR
VERSION : 1.0
// stored: InstanceOfName IEC_TIMER
"IEC_TIMER"
BEGIN
END_DATA_BLOCK

DATA_BLOCK "TimerLengthStation1Port1"   // DB5
{ S7_Optimized_Access := 'TRUE' }
AUTHOR : Simatic
FAMILY : IEC
NAME : IEC_TMR
VERSION : 1.0
// stored: InstanceOfName IEC_TIMER
"IEC_TIMER"
BEGIN
END_DATA_BLOCK

DATA_BLOCK "TimerTagAtHeadStation1Port1"   // DB6
{ S7_Optimized_Access := 'TRUE' }
AUTHOR : Simatic
FAMILY : IEC
NAME : IEC_TMR
VERSION : 1.0
// stored: InstanceOfName IEC_TIMER
"IEC_TIMER"
BEGIN
END_DATA_BLOCK

DATA_BLOCK "IEC_Timer_0_DB_2"   // DB9
{ S7_Optimized_Access := 'TRUE' }
AUTHOR : Simatic
FAMILY : IEC
NAME : IEC_TMR
VERSION : 1.0
// stored: InstanceOfName IEC_TIMER
"IEC_TIMER"
BEGIN
END_DATA_BLOCK

DATA_BLOCK "IEC_Timer_0_DB"   // DB14
{ S7_Optimized_Access := 'TRUE' }
AUTHOR : Simatic
FAMILY : IEC
NAME : IEC_TMR
VERSION : 1.0
// stored: InstanceOfName IEC_TIMER
"IEC_TIMER"
BEGIN
   PT := T#100ms;
END_DATA_BLOCK

DATA_BLOCK "IEC_Timer_0_DB_1"   // DB15
{ S7_Optimized_Access := 'TRUE' }
AUTHOR : Simatic
FAMILY : IEC
NAME : IEC_TMR
VERSION : 1.0
// stored: InstanceOfName IEC_TIMER
"IEC_TIMER"
BEGIN
END_DATA_BLOCK

// folder: (top level)

FUNCTION_BLOCK "Lese"   // FB1, SCL
{ S7_Optimized_Access := 'TRUE' }
VERSION : 0.1
   VAR_OUTPUT
      Wert : Array[0..7] of Byte;
   END_VAR
   VAR
      Adresse : Int;
      EndeAdresse : Int;
   END_VAR
   VAR_TEMP
      i : Int;
      index : Int;
   END_VAR
BEGIN
   #i := 0;
   FOR #index := #Adresse TO #EndeAdresse  DO
       #Wert[#i] := PEEK(area :=16#81,dbNumber:= 0,byteOffset := #index);
       #i := #i + 1;
   END_FOR;
END_FUNCTION_BLOCK

FUNCTION_BLOCK "FB35_IOL_10Byte"   // FB35, STL
TITLE = Schreib-/ Lesebaustein für Balluff RFID System (V1.1)
{ S7_Optimized_Access := 'FALSE' }
AUTHOR : Serrano
FAMILY : Ident
NAME : BISM_IOL
VERSION : 1.0
// Haftungsausschluss:
// *********************
// Der hier kostenlos verfügbare DEMO-Baustein ist ein allgemeingültiges 
// Anwendungsbeispiel. Dieser DEMO-Baustein soll bei der Programmierung und 
// Projektierung von SPS-Anwendungen unterstützen und Lösungsansätze aufzeigen. 
// Ein Anspruch auf Gewährleistung, Fehlerbeseitigung und Update besteht für den 
// Anwender nicht. Die BALLUFF GmbH schließt insbesondere jegliche Haftung für 
// Schäden, die durch den Einsatz dieses DEMO-Bausteins entstehen, ausdrücklich 
// aus! Diese Haftungsbeschränkung gilt nicht bei Verletzungen des Lebens, des 
// Körpers oder der Gesundheit, bei der Haftung nach dem Produkthaftungsgesetz und 
// bei vorsätzlichen Pflichtverletzungen. 
// Prüfen Sie vor dem Einsatz in Anlagen und Maschinen, ob der hier 
// bereitgestellte 
// DEMO Baustein für Ihre Anwendung nutzbar ist!
// Mit dem Einsatz des hier kostenlos vorgelegten S7-Beispiel erkennen Sie die 
// Gewährleistungs- und Haftungsbegrenzung an!
// 
// Disclaimer of Liability
// **********************
// The demo module made available here without cost is a generally accepted 
// example 
// application. This demo module shall support programming and conception of PLC 
// applications and shall provide possible methods of resolution.
// The user is not entitled to claim for warranty, fault clearance and updates. In 
// particular there is excluded any claims against Balluff GmbH for damages that 
// might result from the use of this demo module. Excluded from this limitation of 
// liability shall be (a) those damages that are based on injury to life, limb or 
// health, (b) a liability according to the Produkthaftungsgesetz (German Product 
// Liability Law) and (c) cases of wilful intent.
// Please check if the demo module is serviceable for your application before 
// adapting it in plants and machineries
// By using the S7 sample made available without cost you accept the limitation of 
// warranty and liability!
// 
// 
// BIS M 4XX-045-XXX-07-S4
// IO-Link Schnittstelle (V 1.1)
// 
// Fehlerliste:
// Nr.(HEX)     Bedeutung:          
// -------------------------------------------------------------------------------
//  00          Kein Fehler
//  01          Lesen/ Schreiben nicht möglich, kein Codeträger im Bereich des 
//              Schreib-/ Lesekopfes
//  02          Fehler beim Lesen
//  03          Codeträger wurde während des Lesens aus dem Bereich des Schreib-/
//              Lesekopfes entfernt
//  04          Fehler beim Schreiben
//  05          Codeträger wurde während des Schreibens aus dem Bereich des
//              Schreib-/ Lesekopfes entfernt
//  06          Zugriffsfehler auf den Speicher
//  07          AV-Bit gesetzt, aber Befehlskennung fehlt oder ist ungültig.
//              oder: Anzahl Byte ist 00
//  09          Kabelbruch Schreib-/ Lesekopf oder Kopf nicht angeschlossen
//  0C          EEPROM in der Auswerteeinheit defekt
//  0E          CRC stimmt nicht überein
//  0F          Inhalt der 1. und 2. Bitleiste sind ungleich
//  20          Adressierung des Auftrags liegt außerhalb des Speicherbereichs des 
//              Datenträgers
//  21          Abruf einer Funktion, die beim aktuellen Datenträger nicht möglich 
//              ist
//  30          Überwachungszeit abgelaufen
//  31          ungültiger Auftrag
   VAR_INPUT
      Init : Bool;   // Internal reset and initailisation of FB
      Start : Bool;   // Start command
      Reset : Bool;   // Reset of BIS and FB
      HeadOff : Bool;   // Disable Antenna
      Dynamic : Bool;   // Dynamic read / write function
      HW_ID : Hw_Io;   // HW Identifier address of module
      Command : Int;   // 1=Read;2=Write
      DB_Send : Int;   // Data block write data
      Offset_DBSend : Int;   // Offset of write data
      DB_Receive : Int;   // Data block for read data
      Offset_DBReceive : Int;   // Offset of data read
      StartAddress : Int;   // Start address from data carrier
      NumberOfByte : Int;   // data lenght to be written or read
      Watchdog : S5Time;   // Watchdog of function
      WD_Timer : Timer;   // Watchdog timer
   END_VAR
   VAR_OUTPUT
      READY : Bool;   // Comamnd ready
      Error : Bool;   // Auftrag mit Fehler beendet
      ErrorCode : Int;   // Fehlernummer
      DataCarrierPresent : Bool;   // Data Carrier present
   END_VAR
   VAR
      Busy : Bool;
      EA_Laenge : Int;
      ZeigerByte : Int;   // Aktuelle Lese-/ Schreibadresse
      LaengeByte : Int;   // Anzahl Byte für Lese-/ Schreibzyklus
      ByteProSeite : Int;   // Anzahl maximaler Nutzbyte pro Seite
      Gesamtbyte : Int;   // Gesamtbyte die gelesen bzw. geschrieben werden
      LesenAktiv : Bool;   // Funktion Lesen ist aktiv
      SchreibenAktiv : Bool;   // Funktion Schreiben ist aktiv
      SchreibKonst : Bool;
      ResetAktiv : Bool;   // Funktion rücksetzen ist aktiv
      HeadOffAktiv : Bool;
      Toggle : Bool;   // Letzer Zustand des Toggle-Bit
      ErsterZyklus : Bool;   // Erster Schreib-/ Lesezyklus
      FP_Start : Bool;   // Flankenmerker Start
      IMP_Start : Bool;   // Impulsmerker Start
      FP_Reset : Bool;   // Flankenmerker Reset
      IMP_Reset : Bool;   // Impulsmerker Reset
      FP_CTPR : Bool;   // Flankenmerker Codetag-Present
      IMP_CTPR : Bool;   // Impulsmerker Codetag-Present
      CounterHF : Int;
      SeiteEingang : Array[0..15] of Byte;
      SeiteAusgang : Array[0..15] of Byte;
      Offset : Int;   // Instanz-DB Offset
      OffsetEin : Int;   // Offset Eingangsarray
      OffsetAus : Int;   // Offset Ausgangsarray
      IOAddress : Hw_Io;
   END_VAR
   VAR_TEMP
      InstanzDB : Int;   // Instanz-DB Nummer
      LOG_1 : Bool;   // Logisch 1
      Sp_start : Bool;   // Bei Fehler wird hier der Flankenmerker Start zwischengespeichert
      temp : Byte;   // Temporäre Variable
      schleife : Int;   // Schleifenzähler
      DB_Empf1 : Int;
      DB_Send1 : Int;
      ret : Int;
   END_VAR
BEGIN

REGION Network 1: SPS Anlauf
   // Initialisierung Instanz-Bereich
         AN    #LOG_1;
         S     #LOG_1;
         L     DINO;
         T     #InstanzDB;  // Nummer des Instanz-DB ermitteln
         OPN   DB[ #InstanzDB];
         TAR2;  // Bit-Offset des Instanz-DB
         SLD   8;
         SRD   8;
         L     8;
         /D;  // Offset Instanz-DB
         T     #Offset;
         L     44;
         +I;
         T     #OffsetEin;  // Offset des Eingangsarray
         L     #Offset;
         L     60;
         +I;
         T     #OffsetAus;  // Offset des Ausgangsarray

         L     #HW_ID;
         T     #IOAddress;

         L     10;
         T     #EA_Laenge;  // EA Länge Profibusmodul

         CALL  DPRD_DAT
         ( LADDR   := #IOAddress,
           RET_VAL := #ret,
           RECORD  := #SeiteEingang
         );

         L     #Offset;
         SLW   3;
         LAR1;

         AN    #READY;
         =     #Busy;

         AN    #Init;
         JC    M000;
         L     0;
         T     DBD[AR1, P#30.0];  //DBD30
         T     DBD[AR1, P#34.0];  //DBD34
         T     DBD[AR1, P#38.0];  //DBD38
         T     #ErrorCode;
         S     #READY;
         R     #Error;
         R     #WD_Timer;
         BEU;
END_REGION

REGION Network 2: Kopfabschaltung
   M000: AN    #HeadOff;
         AN    #HeadOffAktiv;
         JC    M015;
         OPN   DB[ #InstanzDB];
         R     #LesenAktiv;
         R     #SchreibenAktiv;
         R     #SchreibKonst;
         R     #Toggle;
         R     #Error;
         L     0;
         T     #ZeigerByte;
         T     #Gesamtbyte;
         T     #ErrorCode;
         L     #OffsetEin;
         SLW   3;
         LAR1;
         A     DIX[AR1, P#0.6];  // HF-bit high
         O     #HeadOffAktiv;
         JC    M001;
         L     #OffsetAus;  // Offset Ausgangsarrey
         SLW   3;
         LAR1;
         L     0;
         T     DIB[AR1, P#0.0];  // Bitleiste rücksetzen
         A     #HeadOff;
         =     DIX[AR1, P#0.5];  // KA-bit setzen
         S     #HeadOffAktiv;
         R     #READY;
         R     #DataCarrierPresent;
         JU    M002;
   M001: L     #OffsetEin;
         SLW   3;
         LAR1;
         A     #HeadOff;
         BEC;
         AN    DIX[AR1, P#0.6];  // HF-bit high
         JC    M003;
         L     #OffsetAus;
         SLW   3;
         LAR1;
         L     0;
         T     DIB[AR1, P#0.0];  // Bitleiste rücksetzen
   M002: L     DIB[AR1, P#0.0];  // 1. Bitleiste
         T     #temp;
         L     #OffsetAus;  // Adresse 2. Bitleiste
         L     #EA_Laenge;
         +I;
         L     1;
         -I;
         SLW   3;
         LAR1;
         L     #temp;
         T     DBB[AR1, P#0.0];
         JU    m100;
   M003: A     #LOG_1;
         R     #HeadOffAktiv;
         A     DIX[AR1, P#0.0];  // Datenträger vorhanden
         =     #DataCarrierPresent;
         BEU;
END_REGION

REGION Network 3: Eingangsdaten einlesen in Empfangs-DB
   // Bitleiste 1 einlesen in Instanz-DB
   M015: OPN   DB[ #InstanzDB];
         L     #OffsetEin;
         SLW   3;
         LAR1;  // Adresse Bitleiste 1 Pointerformat
         L     DBB[AR1, P#0.0];  // Bitleiste 1 einlesen
         T     #temp;

   // Bitleiste 2 einlesen in Instanz-DB
         L     #OffsetEin;
         L     #EA_Laenge;
         +I;
         L     1;
         -I;
         SLW   3;
         LAR1;  // Adresse Bitleiste 2 Pointerformat
         L     DBB[AR1, P#0.0];  // Bitleiste 2 einlesen
         L     #temp;
         <>I;
         BEC;  // Bitleisten unterschiedlich -> BEB
   // Fehlermeldungen abfragen
         AN    DIX[AR1, P#0.3];  //DIX42.3 Fehler vorhanden ?
         O     #Reset;  // oder Reset
         JC    wt1;
         L     #OffsetEin;
         L     1;
         +I;
         SLW   3;
         LAR1;
         L     DBB[AR1, P#0.0];  // Fehlernummer laden
         T     #ErrorCode;
         A     #LOG_1;
         JU    Fehe;
   //
   wt1:  L     #OffsetEin;
         SLW   3;
         LAR1;
   // Datenträger vorhanden
         A     DIX[AR1, P#0.0];  //DIX42.0 Codetag present
         FP    #FP_CTPR;
         =     #IMP_CTPR;
         AN    #IMP_CTPR;  // Wenn keine pos. Flanke CT_Present, dann Sprung
         JC    wt2;
         A     #LOG_1;
         =     #DataCarrierPresent;
         JU    wt3;
   wt2:  L     #OffsetEin;
         SLW   3;
         LAR1;
         AN    DIX[AR1, P#0.0];  //DIX42.0 Wenn Kein CT_Present vom BIS
         R     #DataCarrierPresent;
   wt3:  NOP   0;
END_REGION

REGION Network 4: Auswerteeinheit rücksetzten
         O     #Reset;  // FB-Eingang Reset
         FP    #FP_Reset;  // Hilfsmerker positive Flanke
         =     #IMP_Reset;  // Impulsmerker, ist einen Zyklus "1"
         A     #IMP_Reset;
         S     #ResetAktiv;
         AN    #ResetAktiv;
         JC    M014;
         R     #LesenAktiv;
         R     #SchreibenAktiv;
         R     #SchreibKonst;
         R     #Toggle;
         R     #Error;
         L     0;
         T     #ZeigerByte;
         T     #Gesamtbyte;
         T     #ErrorCode;
         L     #OffsetEin;
         SLW   3;
         TAR1;
         AN    DIX[AR1, P#0.7];  //DIX42.7 Betriebsbereit BIS
         JC    M013;
         L     #OffsetAus;  // Offset Ausgangsarrey
         SLW   3;
         LAR1;
         L     0;
         T     DIB[AR1, P#0.0];  //DIB170 Bitleiste rücksetzen
         S     DIX[AR1, P#0.2];  //DIX170.2 Resetbit setzen
         JU    M012;
   M013: L     #OffsetAus;
         SLW   3;
         LAR1;
         L     0;
         T     DIB[AR1, P#0.0];  //DIB170 Bitleiste rücksetzen
         R     #ResetAktiv;  // Rücksetzen beendet
   M012: L     DIB[AR1, P#0.0];  //DIB170
         T     #temp;
         L     #OffsetAus;  //1. Bitleiste an Ausgangsbyte übergeben
         SLW   3;
         LAR1;
         L     #temp;
         T     DBB[AR1, P#0.0];
         L     #OffsetAus;  // Adresse 2. Bitleiste
         L     #EA_Laenge;
         +I;
         L     1;
         -I;
         SLW   3;
         LAR1;
         L     #temp;
         T     DBB[AR1, P#0.0];
         JU    m100;
   M014: NOP   0;
END_REGION

REGION Network 5: Startauslösung?
         OPN   DB[ #InstanzDB];
         L     #OffsetEin;
         SLW   3;
         LAR1;
         AN    DIX[AR1, P#0.6];  //DIX42.6 Head Fehler
         JC    star;
         O     #ResetAktiv;
         O     #Reset;
         JC    M020;
         L     #CounterHF;  // Zähler um Kabelbruch nicht sofort
         +     1;  // wirksam werden zu lassen.
         T     #CounterHF;
         L     30;
         <>I;
         JC    M020;
         L     #CounterHF;  // Zähler um Kabelbruch nicht sofort
         +     -1;  // wirksam werden zu lassen.
         T     #CounterHF;
         L     9;
         JU    Fehl;
   star: L     0;
         T     #CounterHF;
         AN    #SchreibenAktiv;
         AN    #LesenAktiv;
         AN    #ResetAktiv;
         AN    #SchreibKonst;
         AN    DIX[AR1, P#0.1];  //DIX42.1 Auftrag erkannt und begonnen
         AN    DIX[AR1, P#0.3];  //DIX42.3 Auftrag fehlerhaft/ abgebrochen
         A     DIX[AR1, P#0.7];  //DIX42.7 BIS betriebsbereit
         =     #READY;
         A     #Start;  // FB-Eingang Start
         FP    #FP_Start;  // Hilfsmerker positive Flanke
         =     #IMP_Start;  // Impulsmerker, ist einen Zyklus "1"

         A(;
         O     #IMP_Start;  // Überwachungszeit starten
         O     DIX[AR1, P#0.1];  //DIX42.1 Auftrag angenommen
         );
         AN    DIX[AR1, P#0.3];  //DIX42.3
         AN    #Dynamic;
         L     #Watchdog;
         SD    #WD_Timer;
         AN    #WD_Timer;
         JC    M020;
         L     48;  // Überwachungszeit abgelaufen
         JU    Fehl;
   M020: AN    #LesenAktiv;
         AN    #SchreibenAktiv;
         AN    #SchreibKonst;
         A(;
         AN    #IMP_Start;
         ON    #READY;
         O     DIX[AR1, P#0.1];  //DIX42.1
         );
         BEC;
END_REGION

REGION Network 6: Initialisieren
         O     #LesenAktiv;
         JC    Lese;
         O     #SchreibenAktiv;
         JC    Schr;
         R     #Error;
         OPN   DB[ #InstanzDB];
         L     #OffsetAus;
         SLW   3;
         LAR1;
         L     0;
         T     #ErrorCode;
         T     DIB[AR1, P#0.0];  //DIB170 1. Bitleiste rücksetzen
         A     #LOG_1;
         S     DIX[AR1, P#0.0];  //DIX170.0 Auftrag vorhanden setzten
   // Leseauftrag?
         L     #Command;  // Auftragsnummer laden
         L     1;
         <>I;
         JC    M025;
         S     #LesenAktiv;  // gleich "1" -> Leseauftrag
         L     1;
         T     DIB[AR1, P#1.0];  //DIB171
         L     #Offset_DBReceive;
         T     #ZeigerByte;
         JU    M035;
   // Schreibauftrag?
   M025: L     #Command;  // Auftragsnummer laden
         L     2;
         <>I;
         JC    M026;
         L     2;
         JU    M028;
   M026: L     #Command;
         L     18;  // gleich "12hex" -> CRC Init
         <>I;
         JC    M027;
         L     18;
         JU    M028;

   M027: L     #Command;
         L     50;  // gleich "32hex" -> Konstante Daten
         <>I;
         JC    M030;
         A     #LOG_1;
         S     #SchreibKonst;
         L     50;

   M028: A     #LOG_1;
         S     #SchreibenAktiv;  // gleich "2" -> Schreibauftrag
         T     DIB[AR1, P#1.0];  //DIB171
         L     #Offset_DBSend;
         T     #ZeigerByte;
         JU    M035;

   M030: L     49;  // ungültiger Auftrag
         JU    Fehl;

   // Erster Zyklus
   M035: AN    #ErsterZyklus;
         S     #ErsterZyklus;
         R     #READY;
   // Berechnungen
         L     #EA_Laenge;
         L     2;  // 2 Bitleisten
         -I;
         T     #ByteProSeite;  // Nutzdaten pro Seite

         A     #SchreibKonst;
         JC    M036;

         L     #NumberOfByte;
         T     #Gesamtbyte;
         JU    M037;

   M036: L     0;
         T     #Gesamtbyte;
         L     #DB_Send;
         T     #DB_Send1;
         OPN   DB[ #DB_Send1];
         L     #ZeigerByte;
         SLW   3;
         LAR1;
         L     DBB[AR1, P#0.0];  // 1. Byte Schreibdaten
         T     #temp;
         OPN   DB[ #InstanzDB];
         L     #OffsetAus;
         SLW   3;
         LAR1;
         L     #temp;
         T     DBB[AR1, P#6.0];  // Übertrag in Ausgangspuffer
   M037: NOP   1;
END_REGION

REGION Network 7: Auftrag senden
   // Die erste Bitleiste wird gespiegelt. Auftrag (Lesen, Schreiben) wird 
   // gesendet.
   // Befehlsanhang generieren
         OPN   DB[ #InstanzDB];
         L     #StartAddress;  // Anfang des Datenträgers laden
         CAW;  // Low- und Highbyte tauschen
         T     DIW[AR1, P#2.0];  //DIW172 ins 2. und 3. Byte des Ausgangspuffers schreiben
         L     #NumberOfByte;  // Laenge des Datenträgers laden
         CAW;  // Low- und Highbyte tauschen
         T     DIW[AR1, P#4.0];  //DIW174 ins 4. und 5. Byte des Ausgangspuffers schreiben

   // Erste Bitleiste spiegeln auf letztes Byte
         L     #OffsetAus;
         SLW   3;
         LAR1;
         L     DIB[AR1, P#0.0];  // Bitleiste 1
         T     #temp;
         L     #OffsetAus;
         L     #EA_Laenge;  // Adresse 2. Bitleiste
         +I;
         L     1;
         -I;
         SLW   3;
         LAR1;
         L     #temp;  // 1.Bitleiste kopieren auf 2. Bitleiste
         T     DIB[AR1, P#0.0];
   //    Auftrag schreiben
         JU    m100;
END_REGION

REGION Network 8: Lesen
   Lese: OPN   DB[ #InstanzDB];
         L     #OffsetEin;
         SLW   3;
         LAR1;
         ON    DIX[AR1, P#0.2];  //DIX42.2 Auftrag beendet
         O     DIX[AR1, P#0.3];  //DIX42.3
         BEC;
         AN    #ErsterZyklus;
         A(;
         A     #Toggle;  // Toggle-Zustand letzter Zyklus
         A     DIX[AR1, P#0.5];  //DIX42.5 Aktuelles Toggle-Bit
         O;
         AN    #Toggle;  // Toggle-Zustand letzter Zyklus
         AN    DIX[AR1, P#0.5];  //DIX42.5 Aktuelles Toggle-Bit
         );
         JC    M075;

         L     #ByteProSeite;
         L     #Gesamtbyte;
         <=I;
         JC    M050;
         T     #LaengeByte;  // Nutzdaten kleiner Nutzdaten pro Seite
         JU    M055;
   M050: L     #ByteProSeite;
         T     #LaengeByte;  // Nutzdaten größer gleich Nutzdaten pro Seite
   M055: L     #DB_Receive;
         T     #DB_Empf1;
         L     0;
         T     #schleife;  // Schleifenzähler rücksetzen
   lp3:  L     #schleife;
         L     #OffsetEin;
         +I;
         L     1;
         +I;
         SLW   3;
         LAR1;  // Leseadresse Eingang im Pointerformat
         OPN   DB[ #InstanzDB];
         L     DBB[AR1, P#0.0];
         T     #temp;
         OPN   DB[ #DB_Empf1];
         L     #ZeigerByte;
         L     #schleife;
         +I;
         SLW   3;
         LAR1;  // Zieladresse Empfangs-DB im Pointerformat
         L     #temp;
         T     DBB[AR1, P#0.0];
         L     #schleife;
         L     1;
         +I;
         T     #schleife;
         L     #LaengeByte;
         <I;
         JC    lp3;
         JU    M070;
   M075: L     #Gesamtbyte;
         L     0;
         ==D;
         JC    m090;
         BEU;
END_REGION

REGION Network 9: Schreiben
   Schr: OPN   DB[ #InstanzDB];
         A     DIX[AR1, P#0.2];  //DIX42.2 Auftrag beendet
         JC    M080;
         ON    DIX[AR1, P#0.1];  //DIX42.1 Auftrag begonnen
         O     DIX[AR1, P#0.3];  //DIX42.3 Auftrag Fehler
         BEC;
         A(;
         A     #Toggle;  // Toggle-Zustand letzter Zyklus
         A     DIX[AR1, P#0.5];  //DIX42.5 Aktuelles Toggle-Bit
         O;
         AN    #Toggle;  // Toggle-Zustand letzter Zyklus
         AN    DIX[AR1, P#0.5];  //DIX42.5 Aktuelles Toggle-Bit
         );
         BEC;

         L     #ByteProSeite;
         L     #Gesamtbyte;
         <=I;
         JC    M150;
         T     #LaengeByte;  // Nutzdaten kleiner Nutzdaten pro Seite
         JU    M155;
   M150: L     #ByteProSeite;
         T     #LaengeByte;  // Nutzdaten größer gleich Nutzdaten pro Seite
   //Nutzdaten in Ziel-DB uebertragen
   M155: L     #DB_Send;
         T     #DB_Send1;
         OPN   DB[ #DB_Send1];
         L     0;
         T     #schleife;
   lp5:  L     #ZeigerByte;
         L     #schleife;
         +I;
         SLW   3;
         LAR1;
         OPN   DB[ #DB_Send1];
         L     DBB[AR1, P#0.0];
         T     #temp;
         L     #OffsetAus;
         L     1;
         +I;
         L     #schleife;
         +I;
         SLW   3;
         LAR1;
         L     #temp;
         OPN   DB[ #InstanzDB];
         T     DBB[AR1, P#0.0];
         L     #schleife;
         L     1;
         +I;
         T     #schleife;
         L     #LaengeByte;
         <I;
         JC    lp5;
         JU    M070;
END_REGION

REGION Network 10: schreiben/ lesen
   M070: L     #OffsetEin;
         SLW   3;
         LAR1;
         L     #Gesamtbyte;  //Bytes die noch uebertragen werden müssen
         L     #LaengeByte;  //Bytes die in diesem Zyklus uebertragen wurden
         -I;  //Bytes hinzuaddieren
         T     #Gesamtbyte;

         L     #ZeigerByte;  // Zielbyte erhöhen um Nutzdatenlaenge des E/A-Bereichs
         L     #LaengeByte;
         +I;
         T     #ZeigerByte;

         OPN   DB[ #InstanzDB];
         A     DIX[AR1, P#0.5];  //DIX42.5
         =     #Toggle;  // Toggle-Zustand speichern
         L     #OffsetAus;
         SLW   3;
         LAR1;
         AN    DIX[AR1, P#0.6];
         =     DIX[AR1, P#0.6];  // Toggle-Bit invertieren im Instanz-DB 1. Bitleiste
         L     DIB[AR1, P#0.0];
         T     DIB[AR1, P#9.0];  // Bitleiste 1 kopieren in Bitleiste 2

         A     #ErsterZyklus;
         R     #ErsterZyklus;
         JU    m100;  // Übertragung noch nicht beendet
   M080: L     #OffsetEin;
         SLW   3;
         LAR1;
         AN    DIX[AR1, P#0.2];  // Auftrag Ende
         BEC;
   m090: L     #OffsetAus;
         SLW   3;
         LAR1;
         A     #LOG_1;
         R     #LesenAktiv;
         R     #SchreibenAktiv;
         R     #SchreibKonst;
         R     #Toggle;
         R     DIX[AR1, P#0.0];  // Auftrag vorhanden rücksetzten

         L     #OffsetAus;  // Auftrag vorhanden rücksetzen 1. Bitleiste
         SLW   3;
         LAR1;
         L     0;
         T     DBB[AR1, P#0.0];

         L     #OffsetAus;  // Auftrag vorhanden rücksetzen 2. Bitleiste
         L     #EA_Laenge;
         +I;
         L     1;
         -I;
         SLW   3;
         LAR1;
         L     0;
         T     DBB[AR1, P#0.0];
         JU    m100;
END_REGION

REGION Network 11: Fehler eintragen
   Fehl: T     #ErrorCode;
   Fehe: L     #Offset;
         SLW   3;
         LAR1;
         S     #Error;
         R     #READY;
         A     #FP_Start;
         =     #Sp_start;
         L     0;
         T     DBD[AR1, P#30.0];  //DBD30
         T     DBD[AR1, P#34.0];  //DIB34
         T     DBD[AR1, P#38.0];  //DIB38
         A     #Sp_start;
         =     #FP_Start;
         JU    m090;
END_REGION

REGION Network 12: Ausgangsdaten übertragen
   m100: CALL  DPWR_DAT
         ( LADDR   := #IOAddress,
           RECORD  := #SeiteAusgang,
           RET_VAL := #ret
         );
         BEU;
END_REGION
END_FUNCTION_BLOCK

FUNCTION_BLOCK "BVS_SC"   // FB50, SCL
TITLE = BVS_SC
{ S7_Optimized_Access := 'TRUE' }
AUTHOR : BI-CU
FAMILY : Balluff
VERSION : 1.1
   VAR_INPUT
      Init : Bool;   // Internal reset and initailisation of FB
      CommandStart : Bool;   // Start command
      Cam_ResetWarn : Bool;   // Camera reset warning
      Cam_Stop_Run : Bool;   // Camera stop run
      Cam_Start_Run : Bool;   // Camera start run
      Cam_Trigger : Bool;   // Camera trigger
      Get_Results : Bool;   // Camera command get results
      HW_LADDR : Hw_SubModule;   // Camera hardware address
      Command : Int;   // 1=SwitchApp; 2=GetApp; 3=GetResult; 4=SetInput
      DB_Send : Int;   // Data block camera send data
      Offset_DBSend : Int;   // Offset send data
      DB_Receive : Int;   // Data block camera receive data
      Offset_DBReceive : Int;   // Offset receive data
      Data_Length : Int;   // Data length of set/get commandos
      WD_Time : Time;   // Watchdog of commandos
   END_VAR
   VAR_OUTPUT
      Ready : Bool;   // Comamnd ready and FB ready
      Result_Ready : Bool;   // Camera result ready
      WaitForTrigger : Bool;   // Camera waiting for Trigger
      Cam_Busy : Bool;   // Camera busy
      Cam_Running : Bool;   // Camera running
      Cam_Ready : Bool;   // Camera ready for commandos
      WarnOvertrigg : Bool;   // Camera warning overtriggerd
      WarnOutBufferErr : Bool;   // Camera warning buffer error
      WarnInBufferErr : Bool;   // Camera warning in buffer error
      WarnErrorRate1 : Bool;   // Camera warning
      WarnErrorRate2 : Bool;   // Camera warning
      WarnOverheat : Bool;   // Camera warning
      WarnSystError : Bool;   // Camera warning
      Error : Bool;   // Command or camera Error
      ErrorNumber : Word;   // Error number
   END_VAR
   VAR
      PointerByte : Int;   // Pointer byte
      LengthByte : Int;   // Number of byte for set/get commando
      BytePerPageIn : Int;   // User bytes per page Out
      BytePerPageOut : Int;   // User bytes per page In
      TotalByte : Int;   // Over all byte data to be set/get
      HW_Init : Bool;   // Hardware adresses initialized
      GetCommandActive : Bool;   // Get commado activ
      SetCommandActive : Bool;   // Set commando active
      GComSend : Bool;   // Get Commando send
      ComDatEnd : Bool;   // Comand data transfered
      ResetActive : Bool;   // Reset Active
      ResetWarnActi : Bool;   // Reset warning active
      ResetProc : Bool;   // ResetProcessing
      ToggleOld : Bool;   // Toggle bit last cycle
      FirstCycle : Bool;   // First command cycle
      RE_Start : Bool;   // Rising edge start
      IMP_Start : Bool;   // Rising edge Start
      IMP_Reset : Bool;   // Rising edge Reset
      IMP_Reset_DN : Bool;   // Rising edge Reset done
      IMP_ResWarn : Bool;   // Rising edge Reset
      CAM_Reset : Bool;   // Start camera reset
      ErrorIn : Bool;   // Error bit intern
      WD_TimerIn : Bool;   // Watchdog timer input
      WD_TimerQ : Bool;   // Watchdog timer output
      CO_WaitForTrigger : Bool;   // CAM Out - PLC In waiting for trigger BasAd[50]
      CO_ResultReady : Bool;   // CAM Out - PLC In result ready
      CO_Busy : Bool;   // CAM Out - PLC In busy
      CO_Running : Bool;   // CAM Out - PLC In running
      CO_CamReady : Bool;   // CAM Out - PLC In ready
      CO_Overtriggerd : Bool;   // CAM Out - PLC In overtriggerd
      CO_OutBufferError : Bool;   // CAM Out - PLC In buffer error
      CO_ErrorRate1 : Bool;   // CAM Out - PLC In error rate 1
      CO_ErrorRate2 : Bool;   // CAM Out - PLC In error rate 2
      CO_InputBuffErr : Bool;   // CAM Out - PLC In out buffer error
      CO_Overheat : Bool;   // CAM Out - PLC In overheat
      CO_SystemError : Bool;   // CAM Out - PLC In system error
      CO_HsAcknow : Bool;   // CAM Out - PLC IN handshake acknowledge
      CO_ToggleIn : Bool;   // CAM Out - PLC IN toggle in
      CO_ErrorCom : Bool;   // CAM Out - PLC In communication error
      CO_ComStatus : Byte;   // CAM Out - PLC In command status byte
      CO_OutLengthInt : Int;   // CAM Out - PLC In commando length
      CO_OutArea : Array[0..#OutBuSi] of Byte;   // CAM Out - PLC In data area
      CI_Trigger : Bool;   // PLC Out - CAM In trigger
      CI_R01 : Bool;   // PLC Out - CAM In n.u.
      CI_R02 : Bool;   // PLC Out - CAM In n.u.
      CI_R03 : Bool;   // PLC Out - CAM In n.u.
      CI_ResetWarning : Bool;   // PLC Out - CAM In reset warning
      CI_Reset : Bool;   // PLC Out - CAM In reset
      CI_StartRun : Bool;   // PLC Out - CAM In start run
      CI_StopRun : Bool;   // PLC Out - CAM In stop run
      CI_HsStrobe : Bool;   // PLC Out - CAM In handshake strobe
      CI_ToggleOut : Bool;   // PLC Out - CAM In toggle
      CI_R12 : Bool;   // PLC Out - CAM In n.u.
      CI_R13 : Bool;   // PLC Out - CAM In n.u.
      CI_R14 : Bool;   // PLC Out - CAM In n.u.
      CI_R15 : Bool;   // PLC Out - CAM In n.u.
      CI_R16 : Bool;   // PLC Out - CAM In n.u.
      CI_R17 : Bool;   // PLC Out - CAM In n.u.
      CI_Command : Byte;   // PLC Out - CAM In commando
      CI_InLengInt : Int;   // PLC Out - CAM In length int
      CI_InArea : Array[0..#InBuSi] of Byte;   // PLC Out - CAM In input area
      OldCyComState : Word;   // Commando state last cycle
      WD_Timer : TON_TIME;   // Watchdog timer TON
      PIaddr : UDInt;   // Input address
      PIcount : UInt;   // Input length
      PQaddr : UDInt;   // Output address
      PQcount : UInt;   // Output address
      RetVal_ModulDiag : Int;   // Return value modul diagnosis
      RetVal_RD_Addr : Int;   // Return value read address
      RetVal_RD_DP : Int;   // Return value read input data
      RetVal_WR_DP : Int;   // Return value write output data
      RetVal_Get_ErrID : Word;   // Return value get error ID
      R_TRIG_Reset : R_TRIG;   // R Trigger reset
      R_TRIG_ResetDN : R_TRIG;   // R Trigger reset done
      R_TRIG_ResWarn : R_TRIG;   // R Trigger reset warning
      R_TRIG_CamTrg : R_TRIG;   // R Trigger camera trigger
      R_TRIG_Start : R_TRIG;   // R Trigger camera start
      ErrorCode : DWord;   // Internal camera error code
      CNT_Diag : UInt;   // CNT_Modul Diag
      Diag_Out : DWord;   // Modul Diag
   END_VAR
   VAR_TEMP
      RLO_1 : Bool;   // "1" signal
      tError : Word;   // temp Error Buffer
      tLoop : DInt;   // temp loopcounter
   END_VAR
   VAR CONSTANT
      InBuSi : Int := 512;   // maximum size inputbuffer
      OutBuSi : Int := 512;   // maximum size outputbuffer
   END_VAR
BEGIN
   //=============================================================================
   //Balluff GmbH
   //(c)Copyright (2016) All Rights Reserved
   //-----------------------------------------------------------------------------
   //Library: BalluffVision
   //Tested with: CPU 1214C V4.1
   //Engineering: TIA Portal V13 SP1 
   //Restrictions: -
   //Requirements: PLC (S7-1200 / S7-1500)
   //Functionality: Boolean Camera functions, Camera Commandos
   //-----------------------------------------------------------------------------
   //Change log table:
   //Version  Date       Expert in charge Changes applied
   //01.00.00 29.01.2016 Balluff GmbH BI    First created with TIA V13 SP1
   //=============================================================================
   //
   (*
   Disclaimer of Liability
   **********************
   The demo function block is free of charge and is a universal application 
   example.
   This demo function block shall help program and configure PLC applications and 
   shall provide possible solutions.
   The user is not entitled to claim for warranty, error correction and updates. 
   In 
   particular there is excluded any claims against Balluff GmbH for damages that 
   might result from the use of this demo program. Excluded from this limitation 
   of 
   liability shall be (a) those damages that are based on injury to life, limb or 
   health, (b) a liability according to the Produkthaftungsgesetz (German Product 
   Liability Law) and (c) cases of willful intent.
   Please check if the function block is intended for your application before 
   adapting it in plants and machineries.
   By using the S7 sample, made available free of charge you accept the limitation 
   of 
   warranty and liability!

   Haftungsausschluss:
   *********************
   Der hier kostenlos verfügbare DEMO-Baustein ist ein allgemeingültiges 
   Anwendungsbeispiel. Dieser DEMO-Baustein soll bei der Programmierung und 
   Projektierung von SPS-Anwendungen unterstützen und Lösungsansätze aufzeigen. 
   Ein Anspruch auf Gewährleistung, Fehlerbeseitigung und Update besteht für den 
   Anwender nicht. Die BALLUFF GmbH schließt insbesondere jegliche Haftung für 
   Schäden, die durch den Einsatz dieses DEMO-Bausteins entstehen, ausdrücklich 
   aus! Diese Haftungsbeschränkung gilt nicht bei Verletzungen des Lebens, des 
   Körpers oder der Gesundheit, bei der Haftung nach dem Produkthaftungsgesetz und 
   bei vorsätzlichen Pflichtverletzungen. 
   Prüfen Sie vor dem Einsatz in Anlagen und Maschinen, ob der hier 
   bereitgestellte 
   DEMO Baustein für Ihre Anwendung nutzbar ist!
   Mit dem Einsatz des hier kostenlos vorgelegten S7-Beispiel erkennen Sie die 
   Gewährleistungs- und Haftungsbegrenzung an!
   *)
   //-----------------------------------------------------------------------------
   //FB Init
   //-----------------------------------------------------------------------------
   IF #Init THEN
       #Ready := TRUE;
       #HW_Init := FALSE;
       #GetCommandActive := FALSE;
       #SetCommandActive := FALSE;
       #ResetActive := FALSE;
       #ResetWarnActi := FALSE;
       #ResetProc := FALSE;
       #GComSend := FALSE;
       #ToggleOld := FALSE;
       #FirstCycle := FALSE;
       #ComDatEnd := False;
       #Error := FALSE;
       #ErrorIn := FALSE;
       #CI_HsStrobe := FALSE;
       #CI_ResetWarning := FALSE;
       #CI_Reset := false;
       #PointerByte := 0;
       #BytePerPageIn := 0;
       #BytePerPageOut := 0;
       #TotalByte := 0;
       #ErrorNumber := 0;
       GOTO Job_Reset;
   END_IF;
   //-----------------------------------------------------------------------------
   // Read modul states
   //-----------------------------------------------------------------------------
   #RetVal_ModulDiag := GET_DIAG(MODE := 0, LADDR := #HW_LADDR, CNT_DIAG => #CNT_Diag, DIAG := #Diag_Out);

   //-----------------------------------------------------------------------------
   // Reading PI/PQ addr and data length
   //-----------------------------------------------------------------------------
   IF NOT #HW_Init THEN
       #RetVal_RD_Addr := RD_ADDR(LADDR := #HW_LADDR , PIADDR => #PIaddr, PICount => #PIcount,
                                  PQADDR => #PQaddr, PQCount => #PQcount);
       #HW_Init := TRUE;
   END_IF;
   //-----------------------------------------------------------------------------
   // Cyclic read cam input if HW init done
   //----------------------------------------------------------------------------- 
   IF #HW_Init THEN
       #RetVal_RD_DP := DPRD_DAT(LADDR := #HW_LADDR, RECORD => #CO_OutArea);
   END_IF;

   //-----------------------------------------------------------------------------
   // Comapre bitheader
   //-----------------------------------------------------------------------------
   IF #CO_OutArea[2] <> #CO_OutArea[#PIcount - 1] THEN
       RETURN;
   END_IF;
   //-----------------------------------------------------------------------------
   // Move input bytes to static bits
   //-----------------------------------------------------------------------------
   #CO_WaitForTrigger := #CO_OutArea[0].%X0;
   #CO_ResultReady := #CO_OutArea[0].%X1;
   #CO_Busy := #CO_OutArea[0].%X5;
   #CO_Running := #CO_OutArea[0].%X6;
   #CO_CamReady := #CO_OutArea[0].%X7;
   #CO_Overtriggerd := #CO_OutArea[1].%X0;
   #CO_OutBufferError := #CO_OutArea[1].%X1;
   #CO_Overheat := #CO_OutArea[1].%X6;
   #CO_SystemError := #CO_OutArea[1].%X7;
   #CO_HsAcknow := #CO_OutArea[2].%X0;
   #CO_ToggleIn := #CO_OutArea[2].%X1;
   #CO_ErrorCom := #CO_OutArea[2].%X7;

   //-----------------------------------------------------------------------------
   // Check camera error bit
   //-----------------------------------------------------------------------------
   IF #CO_ErrorCom AND NOT #ErrorIn THEN

       #tError := #CO_OutArea[3];
       #ErrorCode.%B0 := #CO_OutArea[6];
       #ErrorCode.%B1 := #CO_OutArea[7];
       #ErrorCode.%B2 := #CO_OutArea[8];
       #ErrorCode.%B3 := #CO_OutArea[9];
       GOTO Error;
   END_IF;

   //-----------------------------------------------------------------------------
   // Reset camera, start commando with static var #CAM_Reset
   //-----------------------------------------------------------------------------
   #R_TRIG_Reset(CLK := #CAM_Reset,
                 Q => #IMP_Reset);

   IF #IMP_Reset THEN
       #GetCommandActive := FALSE;
       #SetCommandActive := FALSE;
       #ToggleOld := FALSE;
       #Error := FALSE;
       #ErrorIn := FALSE;
       #PointerByte := 0;
       #TotalByte := 0;
       #ErrorNumber := 0;
       #ResetActive := TRUE;
       #ResetProc := TRUE;
       #GComSend := FALSE;
       #Ready := FALSE;
       #ResetWarnActi := FALSE;
       #GComSend := FALSE;
       #ToggleOld := FALSE;
       #FirstCycle := FALSE;
       #ComDatEnd := FALSE;
       #CI_HsStrobe := FALSE;
       #CI_Reset := TRUE;
       #CI_ResetWarning := FALSE;
       GOTO Job_Reset;
   END_IF;
   // Reset active
   IF #ResetActive AND NOT #CO_CamReady THEN
       #ResetActive := FALSE;
       #CI_Reset := False;
   END_IF;

   #R_TRIG_ResetDN(CLK:=#CO_CamReady,
                   Q=>#IMP_Reset_DN);

   IF #IMP_Reset_DN THEN
       #ResetProc := FALSE;
   END_IF;

   //-----------------------------------------------------------------------------
   // Reset Warnbits
   //-----------------------------------------------------------------------------
   #R_TRIG_ResWarn(CLK:=#Cam_ResetWarn,
                   Q=>#IMP_ResWarn);
   IF #IMP_ResWarn THEN
       #Error := FALSE;
       #ErrorIn := FALSE;
       #ErrorNumber := 0;
       #CI_ResetWarning := TRUE;
   END_IF;

   IF NOT #Cam_ResetWarn
       AND NOT #CO_OutBufferError
       AND NOT #CO_InputBuffErr
       AND NOT #CO_ErrorRate1
       AND NOT #CO_ErrorRate2
       AND NOT #CO_Overheat
       THEN
       #CI_ResetWarning := FALSE;
   END_IF;

   //-----------------------------------------------------------------------------
   // Control boolean camera signals
   //-----------------------------------------------------------------------------
   IF #Cam_Start_Run THEN
       #CI_StartRun := TRUE;
       #CI_StopRun := FALSE;
   END_IF;

   IF #Cam_Stop_Run THEN
       #CI_StopRun := TRUE;
       #CI_StartRun := FALSE;
   END_IF;

   #R_TRIG_CamTrg(CLK:=#Cam_Trigger);

   IF #R_TRIG_CamTrg.Q THEN
       #CI_Trigger := TRUE;
   END_IF;

   IF  NOT #Cam_Trigger THEN
       #CI_Trigger := FALSE;
   END_IF;

   //-----------------------------------------------------------------------------
   // Move status-/warnbits to FB output 
   //-----------------------------------------------------------------------------
   #Result_Ready := #CO_ResultReady;
   #WaitForTrigger := #CO_WaitForTrigger;
   #Cam_Busy:= #CO_Busy;
   #Cam_Running := #CO_Running;
   #Cam_Ready := #CO_CamReady;
   #WarnOvertrigg := #CO_Overtriggerd;
   #WarnOutBufferErr := #CO_OutBufferError;
   #WarnErrorRate1 := #CO_ErrorRate1;
   #WarnErrorRate2 := #CO_ErrorRate2;
   #WarnInBufferErr := #CO_InputBuffErr;
   #WarnOverheat := #CO_Overheat;
   #WarnSystError := #CO_SystemError;

   #CI_InArea[0].%X0 := #CI_Trigger;
   #CI_InArea[0].%X4 := #CI_ResetWarning;
   #CI_InArea[0].%X5 := #CI_Reset;
   #CI_InArea[0].%X6 := #CI_StartRun;
   #CI_InArea[0].%X7 := #CI_StopRun;

   //-----------------------------------------------------------------------------
   // FB ready output 
   #Ready := (NOT #GetCommandActive AND
              NOT #SetCommandActive AND
              NOT #CO_HsAcknow AND
              NOT #ResetProc );

   //-----------------------------------------------------------------------------
   // Command Start
   #R_TRIG_Start(CLK := #CommandStart OR #Get_Results ,
                 Q => #IMP_Start);

   //-----------------------------------------------------------------------------
   // Generate error timeout
   //-----------------------------------------------------------------------------
   #WD_TimerIn := #SetCommandActive OR #GetCommandActive;

   #WD_Timer(IN := #WD_TimerIn,
             PT := #WD_Time,
             Q => #WD_TimerQ);

   IF #WD_TimerQ THEN
       #tError := w#16#30;
       GOTO Error;
   END_IF;

   //-----------------------------------------------------------------------------
   // Check HW/Profinet Error when start is set
   //-----------------------------------------------------------------------------
   IF #IMP_Start THEN
       IF #RetVal_RD_Addr <> 0 THEN
           #tError := w#16#40; //Error read address
           GOTO Error;
       END_IF;

       IF #RetVal_RD_DP <> 0 THEN
           #tError := w#16#41; //Error read input data
           GOTO Error;
       END_IF;

       IF #RetVal_WR_DP <> 0 THEN
           #tError := w#16#42; //Error read output data
           GOTO Error;
       END_IF;
   END_IF;

   //-----------------------------------------------------------------------------
   // Generate error data length
   //-----------------------------------------------------------------------------
   IF #IMP_Start AND
       ( #Data_Length < 0) THEN
       #tError := w#16#32;
       GOTO Error;
   END_IF;

   //-----------------------------------------------------------------------------
   // Check controll- bits change - data output
   //-----------------------------------------------------------------------------
   IF #CI_InArea[0] <> #OldCyComState AND NOT #IMP_Start THEN
       GOTO DataOutput;
   END_IF;
   //=============================================================================
   //
   // Camera commandos
   //
   //=============================================================================

   //-----------------------------------------------------------------------------
   // Goto FB end if no job active
   //-----------------------------------------------------------------------------
   IF (NOT #GetCommandActive AND
       NOT #SetCommandActive AND
      (NOT #IMP_Start OR NOT #Ready)) THEN
       RETURN;
   END_IF;

   IF #ComDatEnd THEN  // Check Get or Set
           GOTO CheckHsAck; //CommandEnd;
       ELSIF #GetCommandActive THEN
           GOTO GetCommand;
       ELSIF #SetCommandActive THEN
           GOTO SetCommand;
       END_IF;

   //-----------------------------------------------------------------------------
   // Initialize Command
   //-----------------------------------------------------------------------------
   IF #Get_Results THEN
           #GetCommandActive := TRUE;
           #CI_InArea[2] := 3;
           #CI_InLengInt := 0;
       ELSE

           CASE #Command OF
               1: // Switch Application
                   #SetCommandActive := TRUE;
                   #CI_InArea[2] := 1;
                   #TotalByte := 1;
                   #CI_InLengInt := 1;
               2:  // Get Application ID
                   #GetCommandActive := TRUE;
                   #CI_InArea[2]:= 2;
                   #CI_InLengInt := 0;
               3:  // Get Results
                   #GetCommandActive := TRUE;
                   #CI_InArea[2]:= 3;
                   #CI_InLengInt := 0;
               4:  // Set Inputs       
                   #SetCommandActive := TRUE;
                   #CI_InArea[2] := 4;
                   #TotalByte := #Data_Length;
                   #CI_InLengInt := #Data_Length;
               5:  // Get Camera Info      
                   #GetCommandActive := TRUE;
                   #CI_InArea[2] := 5;
                   #CI_InLengInt := 0;
               6:  // Get Date and Time 
                   #GetCommandActive := TRUE;
                   #CI_InArea[2] := 6;
                   #CI_InLengInt := 0;
               7:  // Set Date and Time      
                   #SetCommandActive := TRUE;
                   #CI_InArea[2] := 7;
                   #TotalByte := 7; 
                   #CI_InLengInt := 7;
               8:  // Set Sequence Number      
                   #SetCommandActive := TRUE;
                   #CI_InArea[2] := 8;
                   #TotalByte := 4; 
                   #CI_InLengInt := 4;
               ELSE
                   #tError := w#16#31;
                   GOTO Error;
               END_CASE;
   END_IF;

   //-----------------------------------------------------------------------------
   // Calculate transmission data length fix bytes + bitheader
   // delete output signals
   //-----------------------------------------------------------------------------
   #BytePerPageIn := UDINT_TO_INT(#PIcount - 7);
   #BytePerPageOut := UDINT_TO_INT(#PQcount - 6);

   #FirstCycle := TRUE;
   #Ready := FALSE;
   #ErrorNumber := 0;
   #Error := FALSE;
   #ErrorIn := FALSE;
   #tError := 0;
   #GComSend := FALSE;

   IF NOT #SetCommandActive THEN
       GOTO GetCommand;
   END_IF;

   //-----------------------------------------------------------------------------
   // Set command, move data from "DB_Send" to camera
   //-----------------------------------------------------------------------------
   SetCommand:;
   IF NOT #FirstCycle AND
       ((#ToggleOld AND #CO_ToggleIn) OR
       (NOT #ToggleOld AND NOT #CO_ToggleIn)) THEN
       RETURN;
   END_IF;

   IF #FirstCycle THEN
       #PointerByte := #Offset_DBSend ;
   END_IF;

   IF #TotalByte <= #BytePerPageOut THEN
           #LengthByte := #TotalByte;
       ELSE
           #LengthByte := #BytePerPageOut;
   END_IF;

   FOR #tLoop := 0 TO #LengthByte - 1 DO 
       #CI_InArea[5 + #tLoop] := PEEK(area := 16#84,
                                      dbNumber := #DB_Send,
                                      byteOffset := #PointerByte + #tLoop);
   END_FOR;

   #CI_HsStrobe := TRUE;

   GOTO CommandEnd;

   GetCommand:;
   //-----------------------------------------------------------------------------
   // Get command, move data from camera to "DB_Receive"
   // Send get commando goto Data output in first cycle  
   //-----------------------------------------------------------------------------
   IF #FirstCycle AND NOT #GComSend THEN
       #GComSend := TRUE;
       #CI_HsStrobe := TRUE;
       GOTO DataOutput;
   END_IF;

   IF #CI_InArea[2] <> #CO_OutArea[3] OR NOT #CO_HsAcknow THEN
       RETURN;
   END_IF;

   IF NOT #FirstCycle AND ((#ToggleOld AND #CO_ToggleIn) OR
       (NOT #ToggleOld AND NOT #CO_ToggleIn)) OR
       (#FirstCycle AND NOT #CO_HsAcknow) THEN
       RETURN;
   END_IF;

   //-----------------------------------------------------------------------------
   // Read camera length byte
   //----------------------------------------------------------------------------- 
   IF #FirstCycle THEN

       #TotalByte := BYTE_TO_INT(#CO_OutArea[5]) +
       SHL(IN := BYTE_TO_INT(#CO_OutArea[4]), N := 8);

       #PointerByte := #Offset_DBReceive;
       IF ( #Data_Length < 0) THEN 
           #tError := 16#32;
           GOTO Error;
       END_IF;
   END_IF;

   IF #TotalByte <= #BytePerPageIn THEN
           #LengthByte := #TotalByte;
          ELSE
           #LengthByte := #BytePerPageIn;
   END_IF;

   FOR #tLoop := 0 TO #LengthByte - 1 DO 
       POKE(area := 16#84,
            dbNumber := #DB_Receive,
            byteOffset := #PointerByte + #tLoop,
            value := #CO_OutArea[6 + #tLoop]);
   END_FOR;
   CommandEnd:;

   //-----------------------------------------------------------------------------
   // Command block end 
   //----------------------------------------------------------------------------- 
   IF NOT #ComDatEnd THEN
       #TotalByte := #TotalByte - #LengthByte;
       #PointerByte := #PointerByte + #LengthByte;
   END_IF;

   IF #TotalByte <= 0 THEN 
       #ComDatEnd := TRUE;
   END_IF;

   IF (#GetCommandActive AND NOT #ComDatEnd)OR
       (NOT #FirstCycle AND #SetCommandActive) THEN
       #CI_ToggleOut := NOT #CI_ToggleOut;
   END_IF;

   #ToggleOld := #CO_ToggleIn;
   #FirstCycle := FALSE;

   CheckHsAck:;

   IF #CO_HsAcknow AND #ComDatEnd THEN
       #ComDatEnd := FALSE;
       #GetCommandActive := FALSE;
       #SetCommandActive := FALSE;
       #CI_HsStrobe := FALSE;
       #CI_ToggleOut := FALSE;
       #ToggleOld := FALSE;

   END_IF;

   //-----------------------------------------------------------------------------
   // Data output fieldbus
   //-----------------------------------------------------------------------------
   DataOutput:;
       // Move bits to byte
       #CI_InArea[0].%X0 := #CI_Trigger;
       #CI_InArea[0].%X4 := #CI_ResetWarning;
       #CI_InArea[0].%X5 := #CI_Reset;
       #CI_InArea[0].%X6 := #CI_StartRun ;
       #CI_InArea[0].%X7 := #CI_StopRun;
       #CI_InArea[1].%X0 := #CI_HsStrobe;
       #CI_InArea[1].%X1 := #CI_ToggleOut;
       #OldCyComState := #CI_InArea[0];

           #CI_InArea[3] := INT_TO_BYTE(SHR(IN := #CI_InLengInt, N := 8));
           #CI_InArea[4] := INT_TO_BYTE(#CI_InLengInt);

           #CI_InArea[#PQcount - 1] := #CI_InArea[1];

   //-----------------------------------------------------------------------------
   // cyclic write plc output to cam input
   //-----------------------------------------------------------------------------

       IF #HW_Init  THEN
           #RetVal_WR_DP := DPWR_DAT(LADDR := #HW_LADDR, RECORD := #CI_InArea);
       END_IF;
       #RetVal_Get_ErrID := GET_ERR_ID();

       IF #RetVal_Get_ErrID <> 0
           AND NOT #Init
           AND NOT #ErrorIn THEN
           #tError := 16#43;
           GOTO Error;
       END_IF;

       RETURN;
   //-----------------------------------------------------------------------------
   // Error output
   //-----------------------------------------------------------------------------
   Error: ;
       #ErrorNumber := #tError;
       #Ready := FALSE;
       #Error := TRUE;
       #ErrorIn := TRUE;

   Job_Reset:  ;
       #GetCommandActive := FALSE;
       #SetCommandActive := FALSE;
       #CI_HsStrobe := FALSE;
       #CI_ToggleOut := FALSE;
       #ComDatEnd := FALSE;
       #ToggleOld := FALSE;
       GOTO DataOutput;
END_FUNCTION_BLOCK

FUNCTION_BLOCK "IO_LINK_MASTER"   // FB50000, SCL
{ S7_Optimized_Access := 'TRUE' }
AUTHOR : Siemens
FAMILY : IO-Link
VERSION : 1.0
   VAR_INPUT
      REQ : Bool;
      ID : Hw_Io;
      RD_WR : Bool;
   END_VAR
   VAR_OUTPUT
      DONE_VALID : Bool;
      BUSY : Bool;
      ERROR : Bool;
      STATUS : DWord := DW#16#00000000;
      SF_STATUS : DWord := DW#16#00000000;
      RD_LEN : Int := INT#0;
   END_VAR
   VAR_IN_OUT
      RECORD_DATA : Array[0..231] of Byte;
   END_VAR
   VAR
      RDREC_Function : RDREC;
      WRREC_Function : WRREC;
      rdrec : Struct
         valid : Bool;
         busy : Bool;
         error : Bool;
         status : DWord := DW#16#00000000;
         len : UInt := UINT#0;
      END_STRUCT;
      wrrec : Struct
         len : UInt := UINT#0;
         done : Bool;
         busy : Bool;
         error : Bool;
         status : DWord := DW#16#00000000;
      END_STRUCT;
      readdata : Array[0..231] of Byte;
      writedata : Array[0..231] of Byte;
      recorddata : Array[0..231] of Byte;
      checktypeID : Struct
         Signature : Word;
         "Version" : Byte;
         NumberofEntry : USInt;
         Entry : Array[1..8] of Byte;
      END_STRUCT;
      R_TRIG_REQ : Bool;
      R_TRIG_REQ_old : Bool;
      sequencecontrol : Int := INT#0;
      typeofrequest : Int := INT#0;
      idpos : DInt := DINT#0;
      readlength : Int := INT#0;
   END_VAR
   VAR_TEMP
      RetVal_MoveBlock : Int;
      i : Int;
      checkID230 : Int;
      checkID220 : Int;
      checkID222 : Int;
   END_VAR
BEGIN
   (*---------------------------------------------------------------------------------------------------------------------
   SIEMENS AG
   ©Copyright 2015. All Rights Reserved.
   -----------------------------------------------------------------------------------------------------------------------
   Limitation of liability
   This software was developed with largest care. However, the author can not guarantee, that the software runs under
   each version of STEP7 on each PLC flawlessly.
   There is no warranty for the software, to the extent permitted by applicable law. The copyright holder provides the
   software "as is" without warranty of any kind, either expressed or implied, including, but not limited to, the implied
   warranties of merchantability and fitness for a particular purpose. The entire risk as to the quality and performance
   of the software is with you. Should the software prove defective, you assume the cost of all necessary servicing,
   repair or correction. In no event unless required by applicable law will the copyright holder be liable to you for
   damages, including any general, special, incidental or consequential damages arising out of the use or inability to
   use the software (including but not limited to loss of data or data being rendered inaccurate or losses sustained by
   you or third parties or a failure of the software to operate with any other programs), even if such holder or other
   party has been advised of the possibility of such damages.
   Permission to use or copy this software for any purpose is hereby granted without fee, provided the above notices are
   retained on all copies. Permission to modify the code and to distribute modified code is granted, provided the above
   notices are retained, and a notice that the code was modified is included with the above copyright notice.
   -----------------------------------------------------------------------------------------------------------------------
   Functionality provided by this source (short description):

   Function block IO_LINK_MASTER - used to read and write the complete configuration of Siemens IO-Link master modules.
   Functionality was described in following documents:
       - SPH IO-Link Integration V1.0 System Description, Chapter 3.6
       - SPH S7+ Modules V1.1 Part 5 IO-Link Integration 1.1, Chapter 4.2

   Status:     Released (tested)
   File name:  IO_LINK_MASTER
   System :    SIMATIC S7-1500
   Version :   1.0
   -----------------------------------------------------------------------------------------------------------------------
   Script to be stored on level ... in project (mark appropriate levels with [x] below)
   [ ] External
   [ ] All levels possible
   [x] Project level
   [ ] Controller level
   [ ] Device level
   [ ] Subobject level
   -----------------------------------------------------------------------------------------------------------------------
   Restrictions, known limitations:
   non
   -----------------------------------------------------------------------------------------------------------------------
   Requirements, prerequisites, External resources used: nothing
   -----------------------------------------------------------------------------------------------------------------------
   Change log table (latest change is at the bottom of the list):
   Version Date Changes applied
   V1.0.0 <2015-02-28> First created with TIA Portal V13 SP1
   ---------------------------------------------------------------------------------------------------------------------*)

   (*---------------------------------------------------------------------------------------------------------------------
   Status of Function (STATUS)
   00000000 = function is ready for request
   00000230 = function checks type of module (read and evaluate data record ID 230)
   00010230 = function reads data record ID 230, if ERROR then please check SF_STATUS too
   00010220 = function reads data record ID 220, if ERROR then please check SF_STATUS too
   00010222 = function reads data record ID 222, if ERROR then please check SF_STATUS too
   00020230 = function writes data record ID 230, if ERROR then please check SF_STATUS too
   00020220 = function writes data record ID 220, if ERROR then please check SF_STATUS too
   00020222 = function writes data record ID 222, if ERROR then please check SF_STATUS too

   Error of Function
   00030000 = unknown type of module, please check SF_STATUS too
   00030001 = undefinied request (neither READ nor WRITE)
   00030002 = no data for restore available
   00030012 = wrong record length of ID230
   00030220 = ID220 not available
   00030222 = ID222 not available
   ---------------------------------------------------------------------------------------------------------------------*)

   (*---------------------------------------------------------------------------------------------------------------------
               NEW REQUEST
   ---------------------------------------------------------------------------------------------------------------------*)            
   // detection rising edge of "REQ"
   #R_TRIG_REQ := #REQ = TRUE AND #R_TRIG_REQ_old = FALSE;
   #R_TRIG_REQ_old := #REQ = TRUE;

   // start new request if not busy
   IF #R_TRIG_REQ = TRUE AND #sequencecontrol = 0 THEN
       // Initialize outputs
       #DONE_VALID := FALSE;
       #BUSY := TRUE;
       #ERROR := FALSE;
       #STATUS := DW#16#00000000;
       #SF_STATUS := DW#16#00000000;
       #RD_LEN := INT#0;

       // Initialize internal tags 
       #idpos := DINT#0;
       #readlength := INT#0;

       // Check if write or read data record (BACKUP / RESTORE)
       IF #RD_WR = TRUE THEN
           #typeofrequest := 2;    // write data record = RESTORE
           #writedata := #RECORD_DATA;    // consistent copy of write data        
       ELSE
           #typeofrequest := 1;    // read data record = BACKUP
           FOR #i := 0 TO 231 DO   // initialize data record before backup
               #readdata[#i] := B#16#0;
           END_FOR;
       END_IF; // set read or write data record

       // Start sequence
       #sequencecontrol := 1;

   ELSE
       ;
   END_IF; // Initializing and setting type of request 

   (*---------------------------------------------------------------------------------------------------------------------
               SEQUENCE CONTROL

        0 = no request in progress
     1..3 = check type of module (Vendor have to be SIEMENS, type have to be IO-LINK)
   10..16 = Read master parameter = BACKUP
   20..26 = Write master parameter = RESTORE
       98 = Function completed and finish without error
       99 = Function aborted with error
   ---------------------------------------------------------------------------------------------------------------------*)
   CASE #sequencecontrol OF
       1:  // read Consistency Check (Index 230d) for check type of module
           // note: consistency check is also used to check type of module (vendor = SIEMENS and type = IO-LINK) 
           #STATUS := DW#16#00000230;
           #RDREC_Function(REQ := TRUE,
                           ID := #ID,
                           INDEX := DINT#230,
                           MLEN := UINT#0,
                           VALID => #rdrec.valid,
                           BUSY => #rdrec.busy,
                           ERROR => #rdrec.error,
                           STATUS => #rdrec.status,
                           LEN => #rdrec.len,
                           RECORD := #checktypeID);

           IF #rdrec.valid = TRUE THEN // ID 230 is available           
               IF #rdrec.len = INT#12 AND BYTE_TO_INT(#checktypeID.Entry[1]) = INT#220 AND BYTE_TO_INT(#checktypeID.Entry[2]) = INT#222 THEN
                   #sequencecontrol := 2;
               ELSIF #rdrec.len <> UINT#12 THEN
                   #ERROR := TRUE;
                   #STATUS := DW#16#00030012;  // set status = wrong record length of ID230
                   #SF_STATUS := DW#16#00000000;
                   #sequencecontrol := 99; // function aborted with error
               ELSIF BYTE_TO_INT(#checktypeID.Entry[1]) <> INT#220 THEN
                   #ERROR := TRUE;
                   #STATUS := DW#16#00030220;  // set status = ID220 not available
                   #SF_STATUS := DW#16#00000000;
                   #sequencecontrol := 99; // function aborted with error
               ELSIF BYTE_TO_INT(#checktypeID.Entry[2]) <> INT#222 THEN
                   #ERROR := TRUE;
                   #STATUS := DW#16#00030222;  // set status = ID222 not available
                   #SF_STATUS := DW#16#00000000;
                   #sequencecontrol := 99; // function aborted with error
               ELSE
                   #ERROR := TRUE;
                   #STATUS := DW#16#00030000;  // set status = unknown type of module, please check REC_STATUS too
                   #SF_STATUS := DW#16#00000000;
                   #sequencecontrol := 99; // function aborted with error                
               END_IF; // check size and entries
           ELSIF #rdrec.error = TRUE THEN  // ID 230 isn't available 
               #ERROR := TRUE;
               #STATUS := DW#16#00030000;  // set status = unknown type of module, please check REC_STATUS too
               #SF_STATUS := #rdrec.status;
               #sequencecontrol := 99; // function aborted with error
           ELSE
               ;
           END_IF;

       2:  // finish check of module    
           #RDREC_Function(REQ := FALSE,
                           ID := #ID,
                           INDEX := DINT#230,
                           MLEN := UINT#0,
                           VALID => #rdrec.valid,
                           BUSY => #rdrec.busy,
                           ERROR => #rdrec.error,
                           STATUS => #rdrec.status,
                           LEN => #rdrec.len,
                           RECORD := #checktypeID);

           IF #rdrec.valid = FALSE THEN
               #sequencecontrol := 3;
           ELSIF #rdrec.error THEN
               #ERROR := TRUE;
               #STATUS := DW#16#00030000;  // set status = unknown type of module, please check REC_STATUS too
               #SF_STATUS := #rdrec.status;
               #sequencecontrol := 99; // function aborted with error
           ELSE
               ;
           END_IF;

       3:  // Check if write or read data record (BACKUP / RESTORE)
           IF #typeofrequest = 1 THEN  // Read master parameter = BACKUP
               #STATUS := DW#16#00010000;  // set status BACKUP
               #sequencecontrol := 10;
           ELSIF #typeofrequest = 2 THEN   // Write master parameter = RESTORE
               #STATUS := DW#16#00020000;  // set status RESTORE
               // Check write data before start writing
               #checkID230 := BYTE_TO_INT(#writedata[0]);    // check for ID230
               #checkID220 := BYTE_TO_INT(#writedata[2]);    // check for ID220
               #checkID222 := BYTE_TO_INT(#writedata[4]);    // check for ID222
               IF #checkID230 <> INT#230 OR #checkID220 <> INT#220 OR #checkID222 <> INT#222 THEN
                   #ERROR := TRUE;
                   #STATUS := DW#16#00030002;  // set status = wrong record length of ID230
                   #SF_STATUS := DW#16#00000000;
                   #sequencecontrol := 99; // function aborted with error
               ELSE
                   #sequencecontrol := 20;
               END_IF;

           ELSE
               #ERROR := TRUE;
               #STATUS := DW#16#00030001;  // set status = undefinied request (neither READ nor WRITE)
               #SF_STATUS := DW#16#00000000;
               #sequencecontrol := 99; // function aborted with error
               ;
           END_IF;

   (*---------------------------------------------------------------------------------------------------------------------
               Read master parameter = BACKUP
   ---------------------------------------------------------------------------------------------------------------------*)
       10: // read Consistency Check = Index 230d
           #STATUS := DW#16#00010230;
           #RDREC_Function(REQ := TRUE,
                           ID := #ID,
                           INDEX := DINT#230,
                           MLEN := UINT#0,
                           VALID => #rdrec.valid,
                           BUSY => #rdrec.busy,
                           ERROR => #rdrec.error,
                           STATUS => #rdrec.status,
                           LEN => #rdrec.len,
                           RECORD := #recorddata);

